REGION Network 1: Клапан регулирующий - 1
   // Зона - 1
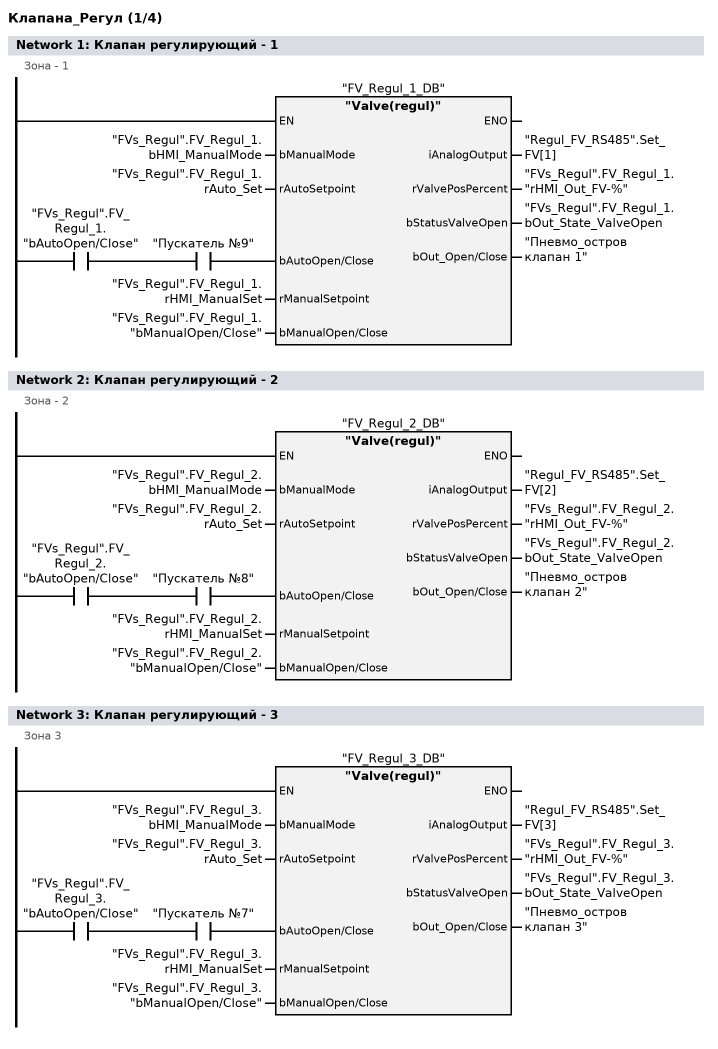
   RUNG wire#powerrail
      "FV_Regul_1_DB"("bAutoOpen/Close" := wire#w1, bManualMode := "FVs_Regul".FV_Regul_1.bHMI_ManualMode, rAutoSetpoint := "FVs_Regul".FV_Regul_1.rAuto_Set, rManualSetpoint := "FVs_Regul".FV_Regul_1.rHMI_ManualSet, "bManualOpen/Close" := "FVs_Regul".FV_Regul_1."bManualOpen/Close", iAnalogOutput => "Regul_FV_RS485".Set_FV[1], rValvePosPercent => "FVs_Regul".FV_Regul_1."rHMI_Out_FV-%", bStatusValveOpen => "FVs_Regul".FV_Regul_1.bOut_State_ValveOpen, "bOut_Open/Close" => "Пневмо_остров клапан 1")
   END_RUNG
   RUNG wire#powerrail
      Contact( "FVs_Regul".FV_Regul_1."bAutoOpen/Close" )
      Contact( "Пускатель №9" )
   END_RUNG wire#w1
   // the same network as SCL:
   "FV_Regul_1_DB"(bManualMode := "FVs_Regul".FV_Regul_1.bHMI_ManualMode,   // "Valve(regul)"
                   rAutoSetpoint := "FVs_Regul".FV_Regul_1.rAuto_Set,
                   "bAutoOpen/Close" := "FVs_Regul".FV_Regul_1."bAutoOpen/Close" AND "Пускатель №9",
                   rManualSetpoint := "FVs_Regul".FV_Regul_1.rHMI_ManualSet,
                   "bManualOpen/Close" := "FVs_Regul".FV_Regul_1."bManualOpen/Close",
                   iAnalogOutput => "Regul_FV_RS485".Set_FV[1],
                   rValvePosPercent => "FVs_Regul".FV_Regul_1."rHMI_Out_FV-%",
                   bStatusValveOpen => "FVs_Regul".FV_Regul_1.bOut_State_ValveOpen,
                   "bOut_Open/Close" => "Пневмо_остров клапан 1");
END_REGION

REGION Network 2: Клапан регулирующий - 2
   // Зона - 2
   RUNG wire#powerrail
      "FV_Regul_2_DB"("bAutoOpen/Close" := wire#w1, bManualMode := "FVs_Regul".FV_Regul_2.bHMI_ManualMode, rAutoSetpoint := "FVs_Regul".FV_Regul_2.rAuto_Set, rManualSetpoint := "FVs_Regul".FV_Regul_2.rHMI_ManualSet, "bManualOpen/Close" := "FVs_Regul".FV_Regul_2."bManualOpen/Close", iAnalogOutput => "Regul_FV_RS485".Set_FV[2], rValvePosPercent => "FVs_Regul".FV_Regul_2."rHMI_Out_FV-%", bStatusValveOpen => "FVs_Regul".FV_Regul_2.bOut_State_ValveOpen, "bOut_Open/Close" => "Пневмо_остров клапан 2")
   END_RUNG
   RUNG wire#powerrail
      Contact( "FVs_Regul".FV_Regul_2."bAutoOpen/Close" )
      Contact( "Пускатель №8" )
   END_RUNG wire#w1
   // the same network as SCL:
   "FV_Regul_2_DB"(bManualMode := "FVs_Regul".FV_Regul_2.bHMI_ManualMode,   // "Valve(regul)"
                   rAutoSetpoint := "FVs_Regul".FV_Regul_2.rAuto_Set,
                   "bAutoOpen/Close" := "FVs_Regul".FV_Regul_2."bAutoOpen/Close" AND "Пускатель №8",
                   rManualSetpoint := "FVs_Regul".FV_Regul_2.rHMI_ManualSet,
                   "bManualOpen/Close" := "FVs_Regul".FV_Regul_2."bManualOpen/Close",
                   iAnalogOutput => "Regul_FV_RS485".Set_FV[2],
                   rValvePosPercent => "FVs_Regul".FV_Regul_2."rHMI_Out_FV-%",
                   bStatusValveOpen => "FVs_Regul".FV_Regul_2.bOut_State_ValveOpen,
                   "bOut_Open/Close" => "Пневмо_остров клапан 2");
END_REGION

REGION Network 3: Клапан регулирующий - 3
   // Зона 3
   RUNG wire#powerrail
      "FV_Regul_3_DB"("bAutoOpen/Close" := wire#w1, bManualMode := "FVs_Regul".FV_Regul_3.bHMI_ManualMode, rAutoSetpoint := "FVs_Regul".FV_Regul_3.rAuto_Set, rManualSetpoint := "FVs_Regul".FV_Regul_3.rHMI_ManualSet, "bManualOpen/Close" := "FVs_Regul".FV_Regul_3."bManualOpen/Close", iAnalogOutput => "Regul_FV_RS485".Set_FV[3], rValvePosPercent => "FVs_Regul".FV_Regul_3."rHMI_Out_FV-%", bStatusValveOpen => "FVs_Regul".FV_Regul_3.bOut_State_ValveOpen, "bOut_Open/Close" => "Пневмо_остров клапан 3")
   END_RUNG
   RUNG wire#powerrail
      Contact( "FVs_Regul".FV_Regul_3."bAutoOpen/Close" )
      Contact( "Пускатель №7" )
   END_RUNG wire#w1
   // the same network as SCL:
   "FV_Regul_3_DB"(bManualMode := "FVs_Regul".FV_Regul_3.bHMI_ManualMode,   // "Valve(regul)"
                   rAutoSetpoint := "FVs_Regul".FV_Regul_3.rAuto_Set,
                   "bAutoOpen/Close" := "FVs_Regul".FV_Regul_3."bAutoOpen/Close" AND "Пускатель №7",
                   rManualSetpoint := "FVs_Regul".FV_Regul_3.rHMI_ManualSet,
                   "bManualOpen/Close" := "FVs_Regul".FV_Regul_3."bManualOpen/Close",
                   iAnalogOutput => "Regul_FV_RS485".Set_FV[3],
                   rValvePosPercent => "FVs_Regul".FV_Regul_3."rHMI_Out_FV-%",
                   bStatusValveOpen => "FVs_Regul".FV_Regul_3.bOut_State_ValveOpen,
                   "bOut_Open/Close" => "Пневмо_остров клапан 3");
END_REGION

REGION Network 4: Клапан регулирующий - 4
   // Зона 4
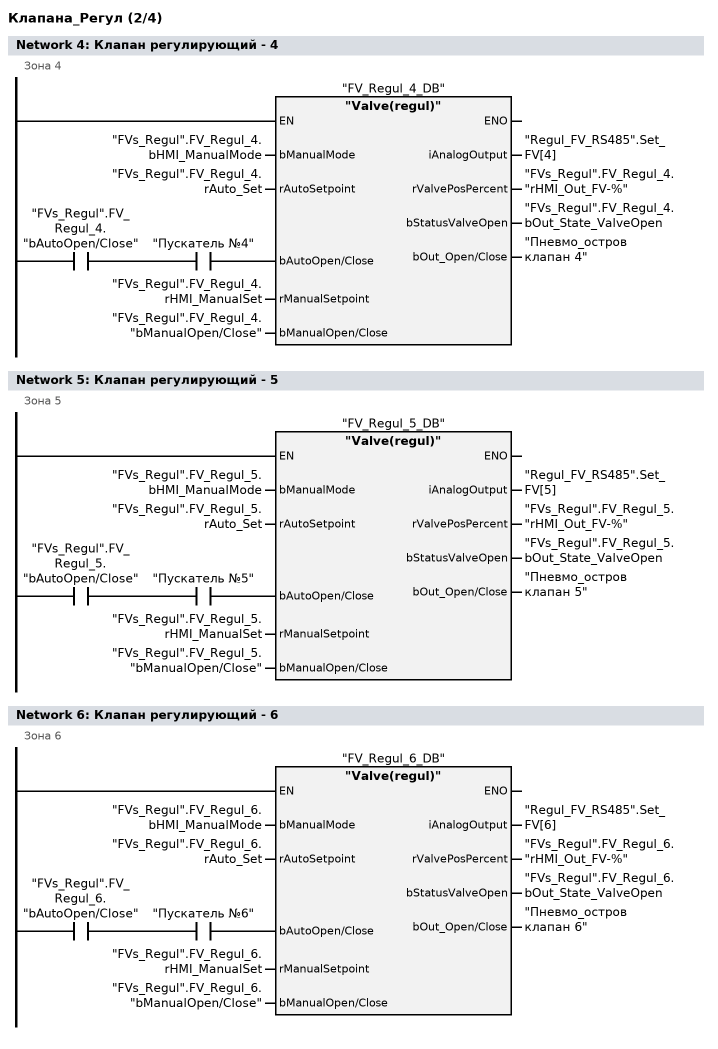
   RUNG wire#powerrail
      "FV_Regul_4_DB"("bAutoOpen/Close" := wire#w1, bManualMode := "FVs_Regul".FV_Regul_4.bHMI_ManualMode, rAutoSetpoint := "FVs_Regul".FV_Regul_4.rAuto_Set, rManualSetpoint := "FVs_Regul".FV_Regul_4.rHMI_ManualSet, "bManualOpen/Close" := "FVs_Regul".FV_Regul_4."bManualOpen/Close", iAnalogOutput => "Regul_FV_RS485".Set_FV[4], rValvePosPercent => "FVs_Regul".FV_Regul_4."rHMI_Out_FV-%", bStatusValveOpen => "FVs_Regul".FV_Regul_4.bOut_State_ValveOpen, "bOut_Open/Close" => "Пневмо_остров клапан 4")
   END_RUNG
   RUNG wire#powerrail
      Contact( "FVs_Regul".FV_Regul_4."bAutoOpen/Close" )
      Contact( "Пускатель №4" )
   END_RUNG wire#w1
   // the same network as SCL:
   "FV_Regul_4_DB"(bManualMode := "FVs_Regul".FV_Regul_4.bHMI_ManualMode,   // "Valve(regul)"
                   rAutoSetpoint := "FVs_Regul".FV_Regul_4.rAuto_Set,
                   "bAutoOpen/Close" := "FVs_Regul".FV_Regul_4."bAutoOpen/Close" AND "Пускатель №4",
                   rManualSetpoint := "FVs_Regul".FV_Regul_4.rHMI_ManualSet,
                   "bManualOpen/Close" := "FVs_Regul".FV_Regul_4."bManualOpen/Close",
                   iAnalogOutput => "Regul_FV_RS485".Set_FV[4],
                   rValvePosPercent => "FVs_Regul".FV_Regul_4."rHMI_Out_FV-%",
                   bStatusValveOpen => "FVs_Regul".FV_Regul_4.bOut_State_ValveOpen,
                   "bOut_Open/Close" => "Пневмо_остров клапан 4");
END_REGION

REGION Network 5: Клапан регулирующий - 5
   // Зона 5
   RUNG wire#powerrail
      "FV_Regul_5_DB"("bAutoOpen/Close" := wire#w1, bManualMode := "FVs_Regul".FV_Regul_5.bHMI_ManualMode, rAutoSetpoint := "FVs_Regul".FV_Regul_5.rAuto_Set, rManualSetpoint := "FVs_Regul".FV_Regul_5.rHMI_ManualSet, "bManualOpen/Close" := "FVs_Regul".FV_Regul_5."bManualOpen/Close", iAnalogOutput => "Regul_FV_RS485".Set_FV[5], rValvePosPercent => "FVs_Regul".FV_Regul_5."rHMI_Out_FV-%", bStatusValveOpen => "FVs_Regul".FV_Regul_5.bOut_State_ValveOpen, "bOut_Open/Close" => "Пневмо_остров клапан 5")
   END_RUNG
   RUNG wire#powerrail
      Contact( "FVs_Regul".FV_Regul_5."bAutoOpen/Close" )
      Contact( "Пускатель №5" )
   END_RUNG wire#w1
   // the same network as SCL:
   "FV_Regul_5_DB"(bManualMode := "FVs_Regul".FV_Regul_5.bHMI_ManualMode,   // "Valve(regul)"
                   rAutoSetpoint := "FVs_Regul".FV_Regul_5.rAuto_Set,
                   "bAutoOpen/Close" := "FVs_Regul".FV_Regul_5."bAutoOpen/Close" AND "Пускатель №5",
                   rManualSetpoint := "FVs_Regul".FV_Regul_5.rHMI_ManualSet,
                   "bManualOpen/Close" := "FVs_Regul".FV_Regul_5."bManualOpen/Close",
                   iAnalogOutput => "Regul_FV_RS485".Set_FV[5],
                   rValvePosPercent => "FVs_Regul".FV_Regul_5."rHMI_Out_FV-%",
                   bStatusValveOpen => "FVs_Regul".FV_Regul_5.bOut_State_ValveOpen,
                   "bOut_Open/Close" => "Пневмо_остров клапан 5");
END_REGION

REGION Network 6: Клапан регулирующий - 6
   // Зона 6
   RUNG wire#powerrail
      "FV_Regul_6_DB"("bAutoOpen/Close" := wire#w1, bManualMode := "FVs_Regul".FV_Regul_6.bHMI_ManualMode, rAutoSetpoint := "FVs_Regul".FV_Regul_6.rAuto_Set, rManualSetpoint := "FVs_Regul".FV_Regul_6.rHMI_ManualSet, "bManualOpen/Close" := "FVs_Regul".FV_Regul_6."bManualOpen/Close", iAnalogOutput => "Regul_FV_RS485".Set_FV[6], rValvePosPercent => "FVs_Regul".FV_Regul_6."rHMI_Out_FV-%", bStatusValveOpen => "FVs_Regul".FV_Regul_6.bOut_State_ValveOpen, "bOut_Open/Close" => "Пневмо_остров клапан 6")
   END_RUNG
   RUNG wire#powerrail
      Contact( "FVs_Regul".FV_Regul_6."bAutoOpen/Close" )
      Contact( "Пускатель №6" )
   END_RUNG wire#w1
   // the same network as SCL:
   "FV_Regul_6_DB"(bManualMode := "FVs_Regul".FV_Regul_6.bHMI_ManualMode,   // "Valve(regul)"
                   rAutoSetpoint := "FVs_Regul".FV_Regul_6.rAuto_Set,
                   "bAutoOpen/Close" := "FVs_Regul".FV_Regul_6."bAutoOpen/Close" AND "Пускатель №6",
                   rManualSetpoint := "FVs_Regul".FV_Regul_6.rHMI_ManualSet,
                   "bManualOpen/Close" := "FVs_Regul".FV_Regul_6."bManualOpen/Close",
                   iAnalogOutput => "Regul_FV_RS485".Set_FV[6],
                   rValvePosPercent => "FVs_Regul".FV_Regul_6."rHMI_Out_FV-%",
                   bStatusValveOpen => "FVs_Regul".FV_Regul_6.bOut_State_ValveOpen,
                   "bOut_Open/Close" => "Пневмо_остров клапан 6");
END_REGION

REGION Network 7: Клапан регулирующий - 7(Холод)
   // Зона 10 - Холод
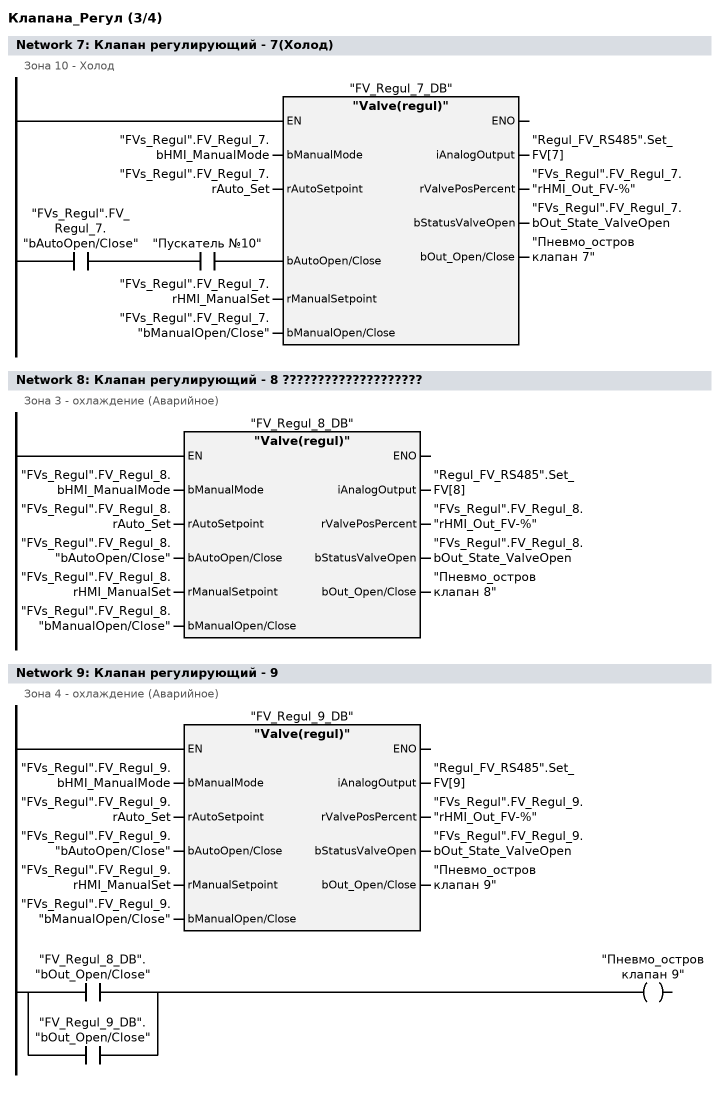
   RUNG wire#powerrail
      "FV_Regul_7_DB"("bAutoOpen/Close" := wire#w1, bManualMode := "FVs_Regul".FV_Regul_7.bHMI_ManualMode, rAutoSetpoint := "FVs_Regul".FV_Regul_7.rAuto_Set, rManualSetpoint := "FVs_Regul".FV_Regul_7.rHMI_ManualSet, "bManualOpen/Close" := "FVs_Regul".FV_Regul_7."bManualOpen/Close", iAnalogOutput => "Regul_FV_RS485".Set_FV[7], rValvePosPercent => "FVs_Regul".FV_Regul_7."rHMI_Out_FV-%", bStatusValveOpen => "FVs_Regul".FV_Regul_7.bOut_State_ValveOpen, "bOut_Open/Close" => "Пневмо_остров клапан 7")
   END_RUNG
   RUNG wire#powerrail
      Contact( "FVs_Regul".FV_Regul_7."bAutoOpen/Close" )
      Contact( "Пускатель №10" )
   END_RUNG wire#w1
   // the same network as SCL:
   "FV_Regul_7_DB"(bManualMode := "FVs_Regul".FV_Regul_7.bHMI_ManualMode,   // "Valve(regul)"
                   rAutoSetpoint := "FVs_Regul".FV_Regul_7.rAuto_Set,
                   "bAutoOpen/Close" := "FVs_Regul".FV_Regul_7."bAutoOpen/Close" AND "Пускатель №10",
                   rManualSetpoint := "FVs_Regul".FV_Regul_7.rHMI_ManualSet,
                   "bManualOpen/Close" := "FVs_Regul".FV_Regul_7."bManualOpen/Close",
                   iAnalogOutput => "Regul_FV_RS485".Set_FV[7],
                   rValvePosPercent => "FVs_Regul".FV_Regul_7."rHMI_Out_FV-%",
                   bStatusValveOpen => "FVs_Regul".FV_Regul_7.bOut_State_ValveOpen,
                   "bOut_Open/Close" => "Пневмо_остров клапан 7");
END_REGION

REGION Network 8: Клапан регулирующий - 8 ????????????????????
   // Зона 3 - охлаждение (Аварийное)
   RUNG wire#powerrail
      "FV_Regul_8_DB"(bManualMode := "FVs_Regul".FV_Regul_8.bHMI_ManualMode, rAutoSetpoint := "FVs_Regul".FV_Regul_8.rAuto_Set, "bAutoOpen/Close" := "FVs_Regul".FV_Regul_8."bAutoOpen/Close", rManualSetpoint := "FVs_Regul".FV_Regul_8.rHMI_ManualSet, "bManualOpen/Close" := "FVs_Regul".FV_Regul_8."bManualOpen/Close", iAnalogOutput => "Regul_FV_RS485".Set_FV[8], rValvePosPercent => "FVs_Regul".FV_Regul_8."rHMI_Out_FV-%", bStatusValveOpen => "FVs_Regul".FV_Regul_8.bOut_State_ValveOpen, "bOut_Open/Close" => "Пневмо_остров клапан 8")
   END_RUNG
   // the same network as SCL:
   "FV_Regul_8_DB"(bManualMode := "FVs_Regul".FV_Regul_8.bHMI_ManualMode,   // "Valve(regul)"
                   rAutoSetpoint := "FVs_Regul".FV_Regul_8.rAuto_Set,
                   "bAutoOpen/Close" := "FVs_Regul".FV_Regul_8."bAutoOpen/Close",
                   rManualSetpoint := "FVs_Regul".FV_Regul_8.rHMI_ManualSet,
                   "bManualOpen/Close" := "FVs_Regul".FV_Regul_8."bManualOpen/Close",
                   iAnalogOutput => "Regul_FV_RS485".Set_FV[8],
                   rValvePosPercent => "FVs_Regul".FV_Regul_8."rHMI_Out_FV-%",
                   bStatusValveOpen => "FVs_Regul".FV_Regul_8.bOut_State_ValveOpen,
                   "bOut_Open/Close" => "Пневмо_остров клапан 8");
END_REGION

REGION Network 9: Клапан регулирующий - 9
   // Зона 4 - охлаждение (Аварийное)
   RUNG wire#powerrail
      "FV_Regul_9_DB"(bManualMode := "FVs_Regul".FV_Regul_9.bHMI_ManualMode, rAutoSetpoint := "FVs_Regul".FV_Regul_9.rAuto_Set, "bAutoOpen/Close" := "FVs_Regul".FV_Regul_9."bAutoOpen/Close", rManualSetpoint := "FVs_Regul".FV_Regul_9.rHMI_ManualSet, "bManualOpen/Close" := "FVs_Regul".FV_Regul_9."bManualOpen/Close", iAnalogOutput => "Regul_FV_RS485".Set_FV[9], rValvePosPercent => "FVs_Regul".FV_Regul_9."rHMI_Out_FV-%", bStatusValveOpen => "FVs_Regul".FV_Regul_9.bOut_State_ValveOpen, "bOut_Open/Close" => "Пневмо_остров клапан 9")
   END_RUNG
   RUNG wire#powerrail
      Contact( "FV_Regul_8_DB"."bOut_Open/Close" )
      wire#w1
      Coil( "Пневмо_остров клапан 9" )
   END_RUNG
   RUNG wire#powerrail
      Contact( "FV_Regul_9_DB"."bOut_Open/Close" )
   END_RUNG wire#w1
   // the same network as SCL:
   "FV_Regul_9_DB"(bManualMode := "FVs_Regul".FV_Regul_9.bHMI_ManualMode,   // "Valve(regul)"
                   rAutoSetpoint := "FVs_Regul".FV_Regul_9.rAuto_Set,
                   "bAutoOpen/Close" := "FVs_Regul".FV_Regul_9."bAutoOpen/Close",
                   rManualSetpoint := "FVs_Regul".FV_Regul_9.rHMI_ManualSet,
                   "bManualOpen/Close" := "FVs_Regul".FV_Regul_9."bManualOpen/Close",
                   iAnalogOutput => "Regul_FV_RS485".Set_FV[9],
                   rValvePosPercent => "FVs_Regul".FV_Regul_9."rHMI_Out_FV-%",
                   bStatusValveOpen => "FVs_Regul".FV_Regul_9.bOut_State_ValveOpen,
                   "bOut_Open/Close" => "Пневмо_остров клапан 9");
   "Пневмо_остров клапан 9" := "FV_Regul_8_DB"."bOut_Open/Close" OR "FV_Regul_9_DB"."bOut_Open/Close";
END_REGION

REGION Network 10: Клапан регулирующий - 10
   // Зона 5 - охлаждение (аварийное)
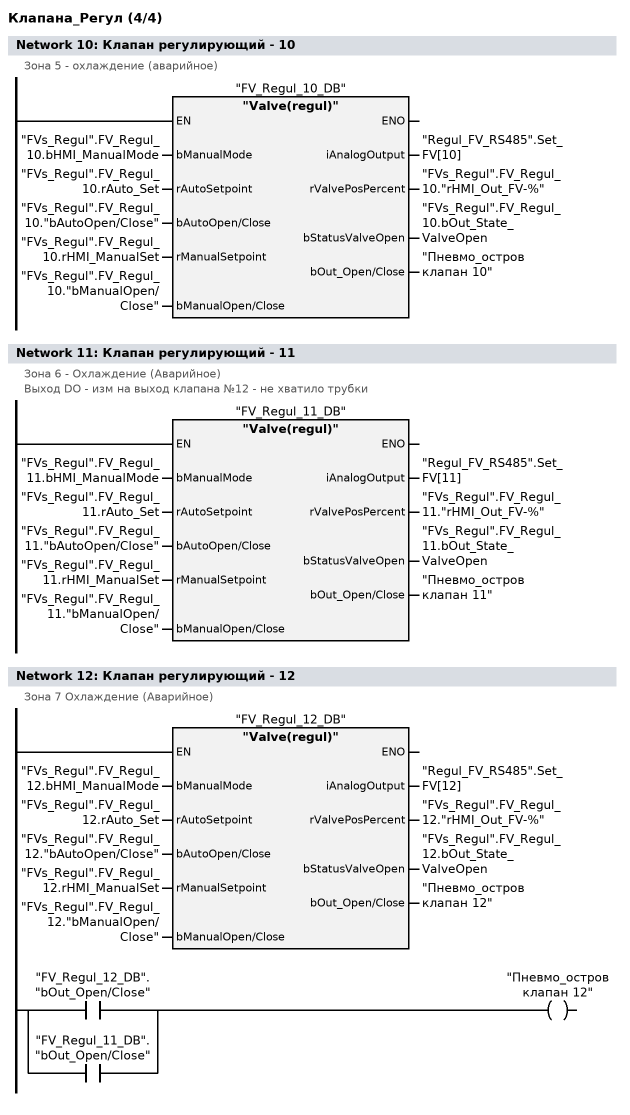
   RUNG wire#powerrail
      "FV_Regul_10_DB"(bManualMode := "FVs_Regul".FV_Regul_10.bHMI_ManualMode, rAutoSetpoint := "FVs_Regul".FV_Regul_10.rAuto_Set, "bAutoOpen/Close" := "FVs_Regul".FV_Regul_10."bAutoOpen/Close", rManualSetpoint := "FVs_Regul".FV_Regul_10.rHMI_ManualSet, "bManualOpen/Close" := "FVs_Regul".FV_Regul_10."bManualOpen/Close", iAnalogOutput => "Regul_FV_RS485".Set_FV[10], rValvePosPercent => "FVs_Regul".FV_Regul_10."rHMI_Out_FV-%", bStatusValveOpen => "FVs_Regul".FV_Regul_10.bOut_State_ValveOpen, "bOut_Open/Close" => "Пневмо_остров клапан 10")
   END_RUNG
   // the same network as SCL:
   "FV_Regul_10_DB"(bManualMode := "FVs_Regul".FV_Regul_10.bHMI_ManualMode,   // "Valve(regul)"
                    rAutoSetpoint := "FVs_Regul".FV_Regul_10.rAuto_Set,
                    "bAutoOpen/Close" := "FVs_Regul".FV_Regul_10."bAutoOpen/Close",
                    rManualSetpoint := "FVs_Regul".FV_Regul_10.rHMI_ManualSet,
                    "bManualOpen/Close" := "FVs_Regul".FV_Regul_10."bManualOpen/Close",
                    iAnalogOutput => "Regul_FV_RS485".Set_FV[10],
                    rValvePosPercent => "FVs_Regul".FV_Regul_10."rHMI_Out_FV-%",
                    bStatusValveOpen => "FVs_Regul".FV_Regul_10.bOut_State_ValveOpen,
                    "bOut_Open/Close" => "Пневмо_остров клапан 10");
END_REGION

REGION Network 11: Клапан регулирующий - 11
   // Зона 6 - Охлаждение (Аварийное)
   // Выход DO - изм на выход клапана №12 - не хватило трубки
   RUNG wire#powerrail
      "FV_Regul_11_DB"(bManualMode := "FVs_Regul".FV_Regul_11.bHMI_ManualMode, rAutoSetpoint := "FVs_Regul".FV_Regul_11.rAuto_Set, "bAutoOpen/Close" := "FVs_Regul".FV_Regul_11."bAutoOpen/Close", rManualSetpoint := "FVs_Regul".FV_Regul_11.rHMI_ManualSet, "bManualOpen/Close" := "FVs_Regul".FV_Regul_11."bManualOpen/Close", iAnalogOutput => "Regul_FV_RS485".Set_FV[11], rValvePosPercent => "FVs_Regul".FV_Regul_11."rHMI_Out_FV-%", bStatusValveOpen => "FVs_Regul".FV_Regul_11.bOut_State_ValveOpen, "bOut_Open/Close" => "Пневмо_остров клапан 11")
   END_RUNG
   // the same network as SCL:
   "FV_Regul_11_DB"(bManualMode := "FVs_Regul".FV_Regul_11.bHMI_ManualMode,   // "Valve(regul)"
                    rAutoSetpoint := "FVs_Regul".FV_Regul_11.rAuto_Set,
                    "bAutoOpen/Close" := "FVs_Regul".FV_Regul_11."bAutoOpen/Close",
                    rManualSetpoint := "FVs_Regul".FV_Regul_11.rHMI_ManualSet,
                    "bManualOpen/Close" := "FVs_Regul".FV_Regul_11."bManualOpen/Close",
                    iAnalogOutput => "Regul_FV_RS485".Set_FV[11],
                    rValvePosPercent => "FVs_Regul".FV_Regul_11."rHMI_Out_FV-%",
                    bStatusValveOpen => "FVs_Regul".FV_Regul_11.bOut_State_ValveOpen,
                    "bOut_Open/Close" => "Пневмо_остров клапан 11");
END_REGION

REGION Network 12: Клапан регулирующий - 12
   // Зона 7 Охлаждение (Аварийное)
   RUNG wire#powerrail
      "FV_Regul_12_DB"(bManualMode := "FVs_Regul".FV_Regul_12.bHMI_ManualMode, rAutoSetpoint := "FVs_Regul".FV_Regul_12.rAuto_Set, "bAutoOpen/Close" := "FVs_Regul".FV_Regul_12."bAutoOpen/Close", rManualSetpoint := "FVs_Regul".FV_Regul_12.rHMI_ManualSet, "bManualOpen/Close" := "FVs_Regul".FV_Regul_12."bManualOpen/Close", iAnalogOutput => "Regul_FV_RS485".Set_FV[12], rValvePosPercent => "FVs_Regul".FV_Regul_12."rHMI_Out_FV-%", bStatusValveOpen => "FVs_Regul".FV_Regul_12.bOut_State_ValveOpen, "bOut_Open/Close" => "Пневмо_остров клапан 12")
   END_RUNG
   RUNG wire#powerrail
      Contact( "FV_Regul_12_DB"."bOut_Open/Close" )
      wire#w1
      Coil( "Пневмо_остров клапан 12" )
   END_RUNG
   RUNG wire#powerrail
      Contact( "FV_Regul_11_DB"."bOut_Open/Close" )
   END_RUNG wire#w1
   // the same network as SCL:
   "FV_Regul_12_DB"(bManualMode := "FVs_Regul".FV_Regul_12.bHMI_ManualMode,   // "Valve(regul)"
                    rAutoSetpoint := "FVs_Regul".FV_Regul_12.rAuto_Set,
                    "bAutoOpen/Close" := "FVs_Regul".FV_Regul_12."bAutoOpen/Close",
                    rManualSetpoint := "FVs_Regul".FV_Regul_12.rHMI_ManualSet,
                    "bManualOpen/Close" := "FVs_Regul".FV_Regul_12."bManualOpen/Close",
                    iAnalogOutput => "Regul_FV_RS485".Set_FV[12],
                    rValvePosPercent => "FVs_Regul".FV_Regul_12."rHMI_Out_FV-%",
                    bStatusValveOpen => "FVs_Regul".FV_Regul_12.bOut_State_ValveOpen,
                    "bOut_Open/Close" => "Пневмо_остров клапан 12");
   "Пневмо_остров клапан 12" := "FV_Regul_12_DB"."bOut_Open/Close" OR "FV_Regul_11_DB"."bOut_Open/Close";
END_REGION

REGION Network 13 (SCL): Клапана регулирующие ручной режим с вфходом DO
   // Для перевода клапана регулирующего в ручной режим должен перейти по сигналу от ручного режим с клапана DO, т.е. для работы клапана регулирующего необходим сигнал DO
   (*"FVs_o/p".FV_1.bManualMode := "FVs_Regul".FV_Regul_1.bHMI_ManualMode;
   "FVs_o/p".FV_2.bManualMode := "FVs_Regul".FV_Regul_2.bHMI_ManualMode;
   "FVs_o/p".FV_3.bManualMode := "FVs_Regul".FV_Regul_3.bHMI_ManualMode;
   "FVs_o/p".FV_4.bManualMode := "FVs_Regul".FV_Regul_5.bHMI_ManualMode;
   *)
END_REGION
END_FUNCTION

FUNCTION "Зоны Пастеризации_Контроль" : Void   // FC3, LAD
{ S7_Optimized_Access := 'TRUE' }
VERSION : 0.1
BEGIN

REGION Network 1: Зона 1(Нагрев)
   // Зона 1
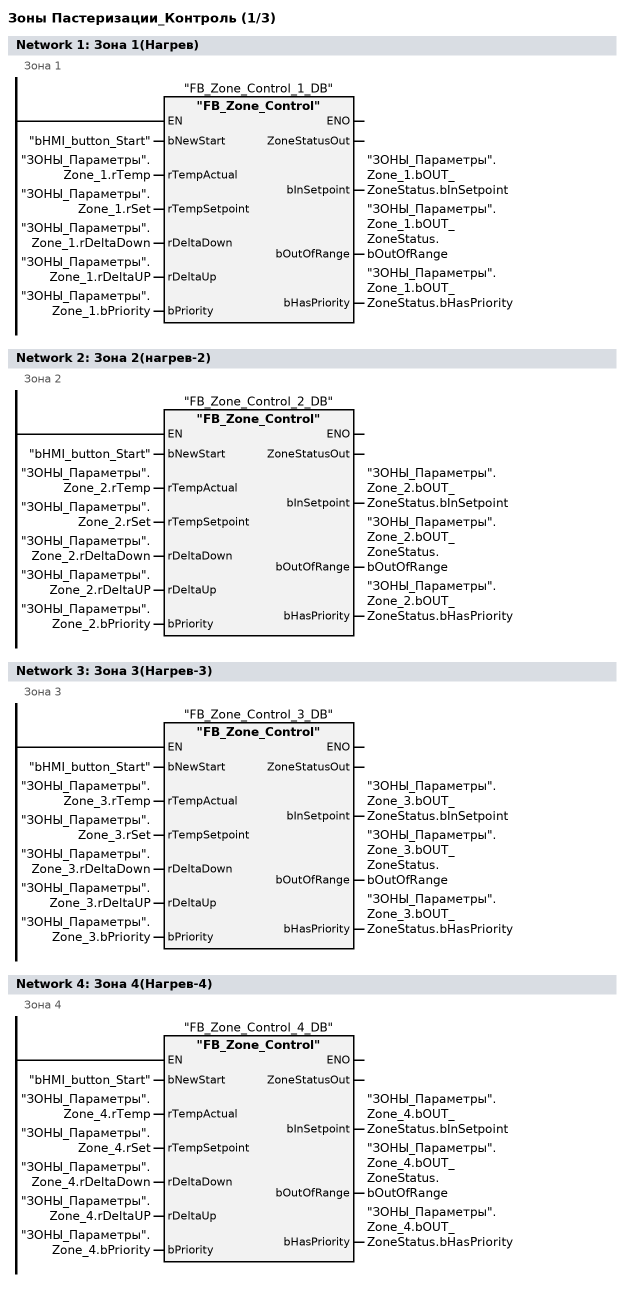
   RUNG wire#powerrail
      "FB_Zone_Control_1_DB"(bNewStart := "bHMI_button_Start", rTempActual := "ЗОНЫ_Параметры".Zone_1.rTemp, rTempSetpoint := "ЗОНЫ_Параметры".Zone_1.rSet, rDeltaDown := "ЗОНЫ_Параметры".Zone_1.rDeltaDown, rDeltaUp := "ЗОНЫ_Параметры".Zone_1.rDeltaUP, bPriority := "ЗОНЫ_Параметры".Zone_1.bPriority, ZoneStatusOut =>, bInSetpoint => "ЗОНЫ_Параметры".Zone_1.bOUT_ZoneStatus.bInSetpoint, bOutOfRange => "ЗОНЫ_Параметры".Zone_1.bOUT_ZoneStatus.bOutOfRange, bHasPriority => "ЗОНЫ_Параметры".Zone_1.bOUT_ZoneStatus.bHasPriority)
   END_RUNG
   // the same network as SCL:
   "FB_Zone_Control_1_DB"(bNewStart := "bHMI_button_Start",   // "FB_Zone_Control"
                          rTempActual := "ЗОНЫ_Параметры".Zone_1.rTemp,
                          rTempSetpoint := "ЗОНЫ_Параметры".Zone_1.rSet,
                          rDeltaDown := "ЗОНЫ_Параметры".Zone_1.rDeltaDown,
                          rDeltaUp := "ЗОНЫ_Параметры".Zone_1.rDeltaUP,
                          bPriority := "ЗОНЫ_Параметры".Zone_1.bPriority,
                          bInSetpoint => "ЗОНЫ_Параметры".Zone_1.bOUT_ZoneStatus.bInSetpoint,
                          bOutOfRange => "ЗОНЫ_Параметры".Zone_1.bOUT_ZoneStatus.bOutOfRange,
                          bHasPriority => "ЗОНЫ_Параметры".Zone_1.bOUT_ZoneStatus.bHasPriority);
END_REGION

REGION Network 2: Зона 2(нагрев-2)
   // Зона 2
   RUNG wire#powerrail
      "FB_Zone_Control_2_DB"(bNewStart := "bHMI_button_Start", rTempActual := "ЗОНЫ_Параметры".Zone_2.rTemp, rTempSetpoint := "ЗОНЫ_Параметры".Zone_2.rSet, rDeltaDown := "ЗОНЫ_Параметры".Zone_2.rDeltaDown, rDeltaUp := "ЗОНЫ_Параметры".Zone_2.rDeltaUP, bPriority := "ЗОНЫ_Параметры".Zone_2.bPriority, ZoneStatusOut =>, bInSetpoint => "ЗОНЫ_Параметры".Zone_2.bOUT_ZoneStatus.bInSetpoint, bOutOfRange => "ЗОНЫ_Параметры".Zone_2.bOUT_ZoneStatus.bOutOfRange, bHasPriority => "ЗОНЫ_Параметры".Zone_2.bOUT_ZoneStatus.bHasPriority)
   END_RUNG
   // the same network as SCL:
   "FB_Zone_Control_2_DB"(bNewStart := "bHMI_button_Start",   // "FB_Zone_Control"
                          rTempActual := "ЗОНЫ_Параметры".Zone_2.rTemp,
                          rTempSetpoint := "ЗОНЫ_Параметры".Zone_2.rSet,
                          rDeltaDown := "ЗОНЫ_Параметры".Zone_2.rDeltaDown,
                          rDeltaUp := "ЗОНЫ_Параметры".Zone_2.rDeltaUP,
                          bPriority := "ЗОНЫ_Параметры".Zone_2.bPriority,
                          bInSetpoint => "ЗОНЫ_Параметры".Zone_2.bOUT_ZoneStatus.bInSetpoint,
                          bOutOfRange => "ЗОНЫ_Параметры".Zone_2.bOUT_ZoneStatus.bOutOfRange,
                          bHasPriority => "ЗОНЫ_Параметры".Zone_2.bOUT_ZoneStatus.bHasPriority);
END_REGION

REGION Network 3: Зона 3(Нагрев-3)
   // Зона 3
   RUNG wire#powerrail
      "FB_Zone_Control_3_DB"(bNewStart := "bHMI_button_Start", rTempActual := "ЗОНЫ_Параметры".Zone_3.rTemp, rTempSetpoint := "ЗОНЫ_Параметры".Zone_3.rSet, rDeltaDown := "ЗОНЫ_Параметры".Zone_3.rDeltaDown, rDeltaUp := "ЗОНЫ_Параметры".Zone_3.rDeltaUP, bPriority := "ЗОНЫ_Параметры".Zone_3.bPriority, ZoneStatusOut =>, bInSetpoint => "ЗОНЫ_Параметры".Zone_3.bOUT_ZoneStatus.bInSetpoint, bOutOfRange => "ЗОНЫ_Параметры".Zone_3.bOUT_ZoneStatus.bOutOfRange, bHasPriority => "ЗОНЫ_Параметры".Zone_3.bOUT_ZoneStatus.bHasPriority)
   END_RUNG
   // the same network as SCL:
   "FB_Zone_Control_3_DB"(bNewStart := "bHMI_button_Start",   // "FB_Zone_Control"
                          rTempActual := "ЗОНЫ_Параметры".Zone_3.rTemp,
                          rTempSetpoint := "ЗОНЫ_Параметры".Zone_3.rSet,
                          rDeltaDown := "ЗОНЫ_Параметры".Zone_3.rDeltaDown,
                          rDeltaUp := "ЗОНЫ_Параметры".Zone_3.rDeltaUP,
                          bPriority := "ЗОНЫ_Параметры".Zone_3.bPriority,
                          bInSetpoint => "ЗОНЫ_Параметры".Zone_3.bOUT_ZoneStatus.bInSetpoint,
                          bOutOfRange => "ЗОНЫ_Параметры".Zone_3.bOUT_ZoneStatus.bOutOfRange,
                          bHasPriority => "ЗОНЫ_Параметры".Zone_3.bOUT_ZoneStatus.bHasPriority);
END_REGION

REGION Network 4: Зона 4(Нагрев-4)
   // Зона 4
   RUNG wire#powerrail
      "FB_Zone_Control_4_DB"(bNewStart := "bHMI_button_Start", rTempActual := "ЗОНЫ_Параметры".Zone_4.rTemp, rTempSetpoint := "ЗОНЫ_Параметры".Zone_4.rSet, rDeltaDown := "ЗОНЫ_Параметры".Zone_4.rDeltaDown, rDeltaUp := "ЗОНЫ_Параметры".Zone_4.rDeltaUP, bPriority := "ЗОНЫ_Параметры".Zone_4.bPriority, ZoneStatusOut =>, bInSetpoint => "ЗОНЫ_Параметры".Zone_4.bOUT_ZoneStatus.bInSetpoint, bOutOfRange => "ЗОНЫ_Параметры".Zone_4.bOUT_ZoneStatus.bOutOfRange, bHasPriority => "ЗОНЫ_Параметры".Zone_4.bOUT_ZoneStatus.bHasPriority)
   END_RUNG
   // the same network as SCL:
   "FB_Zone_Control_4_DB"(bNewStart := "bHMI_button_Start",   // "FB_Zone_Control"
                          rTempActual := "ЗОНЫ_Параметры".Zone_4.rTemp,
                          rTempSetpoint := "ЗОНЫ_Параметры".Zone_4.rSet,
                          rDeltaDown := "ЗОНЫ_Параметры".Zone_4.rDeltaDown,
                          rDeltaUp := "ЗОНЫ_Параметры".Zone_4.rDeltaUP,
                          bPriority := "ЗОНЫ_Параметры".Zone_4.bPriority,
                          bInSetpoint => "ЗОНЫ_Параметры".Zone_4.bOUT_ZoneStatus.bInSetpoint,
                          bOutOfRange => "ЗОНЫ_Параметры".Zone_4.bOUT_ZoneStatus.bOutOfRange,
                          bHasPriority => "ЗОНЫ_Параметры".Zone_4.bOUT_ZoneStatus.bHasPriority);
END_REGION

REGION Network 5: Зона 5(Выдержка-1)
   // Зона 5
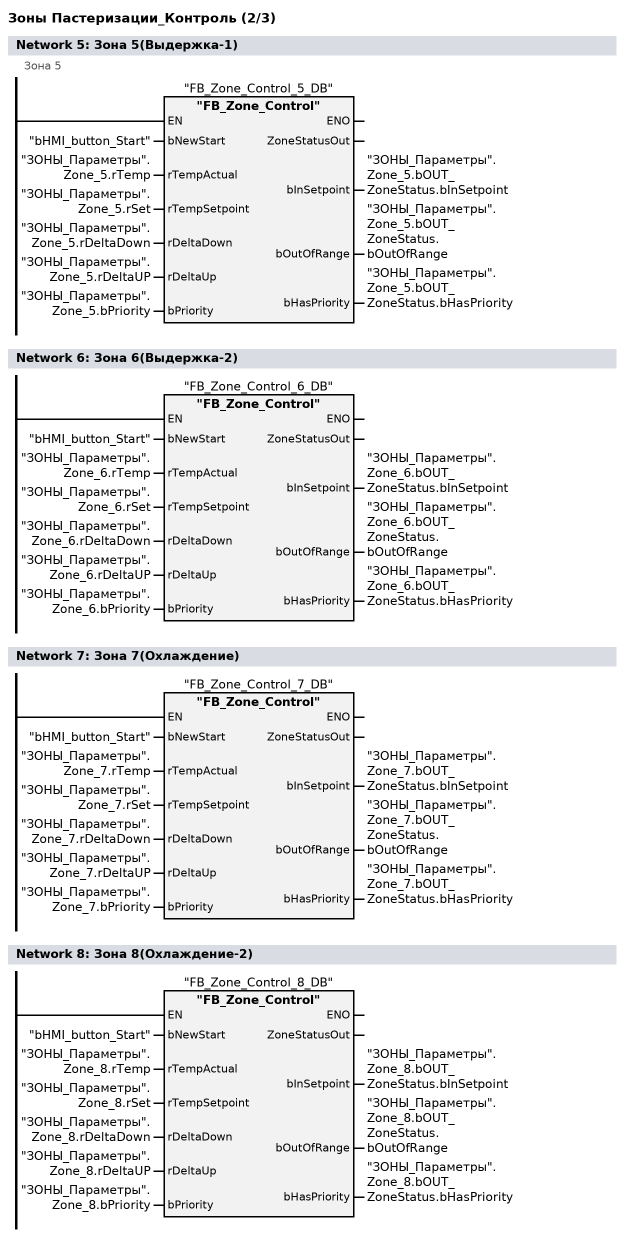
   RUNG wire#powerrail
      "FB_Zone_Control_5_DB"(bNewStart := "bHMI_button_Start", rTempActual := "ЗОНЫ_Параметры".Zone_5.rTemp, rTempSetpoint := "ЗОНЫ_Параметры".Zone_5.rSet, rDeltaDown := "ЗОНЫ_Параметры".Zone_5.rDeltaDown, rDeltaUp := "ЗОНЫ_Параметры".Zone_5.rDeltaUP, bPriority := "ЗОНЫ_Параметры".Zone_5.bPriority, ZoneStatusOut =>, bInSetpoint => "ЗОНЫ_Параметры".Zone_5.bOUT_ZoneStatus.bInSetpoint, bOutOfRange => "ЗОНЫ_Параметры".Zone_5.bOUT_ZoneStatus.bOutOfRange, bHasPriority => "ЗОНЫ_Параметры".Zone_5.bOUT_ZoneStatus.bHasPriority)
   END_RUNG
   // the same network as SCL:
   "FB_Zone_Control_5_DB"(bNewStart := "bHMI_button_Start",   // "FB_Zone_Control"
                          rTempActual := "ЗОНЫ_Параметры".Zone_5.rTemp,
                          rTempSetpoint := "ЗОНЫ_Параметры".Zone_5.rSet,
                          rDeltaDown := "ЗОНЫ_Параметры".Zone_5.rDeltaDown,
                          rDeltaUp := "ЗОНЫ_Параметры".Zone_5.rDeltaUP,
                          bPriority := "ЗОНЫ_Параметры".Zone_5.bPriority,
                          bInSetpoint => "ЗОНЫ_Параметры".Zone_5.bOUT_ZoneStatus.bInSetpoint,
                          bOutOfRange => "ЗОНЫ_Параметры".Zone_5.bOUT_ZoneStatus.bOutOfRange,
                          bHasPriority => "ЗОНЫ_Параметры".Zone_5.bOUT_ZoneStatus.bHasPriority);
END_REGION

REGION Network 6: Зона 6(Выдержка-2)
   RUNG wire#powerrail
      "FB_Zone_Control_6_DB"(bNewStart := "bHMI_button_Start", rTempActual := "ЗОНЫ_Параметры".Zone_6.rTemp, rTempSetpoint := "ЗОНЫ_Параметры".Zone_6.rSet, rDeltaDown := "ЗОНЫ_Параметры".Zone_6.rDeltaDown, rDeltaUp := "ЗОНЫ_Параметры".Zone_6.rDeltaUP, bPriority := "ЗОНЫ_Параметры".Zone_6.bPriority, ZoneStatusOut =>, bInSetpoint => "ЗОНЫ_Параметры".Zone_6.bOUT_ZoneStatus.bInSetpoint, bOutOfRange => "ЗОНЫ_Параметры".Zone_6.bOUT_ZoneStatus.bOutOfRange, bHasPriority => "ЗОНЫ_Параметры".Zone_6.bOUT_ZoneStatus.bHasPriority)
   END_RUNG
   // the same network as SCL:
   "FB_Zone_Control_6_DB"(bNewStart := "bHMI_button_Start",   // "FB_Zone_Control"
                          rTempActual := "ЗОНЫ_Параметры".Zone_6.rTemp,
                          rTempSetpoint := "ЗОНЫ_Параметры".Zone_6.rSet,
                          rDeltaDown := "ЗОНЫ_Параметры".Zone_6.rDeltaDown,
                          rDeltaUp := "ЗОНЫ_Параметры".Zone_6.rDeltaUP,
                          bPriority := "ЗОНЫ_Параметры".Zone_6.bPriority,
                          bInSetpoint => "ЗОНЫ_Параметры".Zone_6.bOUT_ZoneStatus.bInSetpoint,
                          bOutOfRange => "ЗОНЫ_Параметры".Zone_6.bOUT_ZoneStatus.bOutOfRange,
                          bHasPriority => "ЗОНЫ_Параметры".Zone_6.bOUT_ZoneStatus.bHasPriority);
END_REGION

REGION Network 7: Зона 7(Охлаждение)
   RUNG wire#powerrail
      "FB_Zone_Control_7_DB"(bNewStart := "bHMI_button_Start", rTempActual := "ЗОНЫ_Параметры".Zone_7.rTemp, rTempSetpoint := "ЗОНЫ_Параметры".Zone_7.rSet, rDeltaDown := "ЗОНЫ_Параметры".Zone_7.rDeltaDown, rDeltaUp := "ЗОНЫ_Параметры".Zone_7.rDeltaUP, bPriority := "ЗОНЫ_Параметры".Zone_7.bPriority, ZoneStatusOut =>, bInSetpoint => "ЗОНЫ_Параметры".Zone_7.bOUT_ZoneStatus.bInSetpoint, bOutOfRange => "ЗОНЫ_Параметры".Zone_7.bOUT_ZoneStatus.bOutOfRange, bHasPriority => "ЗОНЫ_Параметры".Zone_7.bOUT_ZoneStatus.bHasPriority)
   END_RUNG
   // the same network as SCL:
   "FB_Zone_Control_7_DB"(bNewStart := "bHMI_button_Start",   // "FB_Zone_Control"
                          rTempActual := "ЗОНЫ_Параметры".Zone_7.rTemp,
                          rTempSetpoint := "ЗОНЫ_Параметры".Zone_7.rSet,
                          rDeltaDown := "ЗОНЫ_Параметры".Zone_7.rDeltaDown,
                          rDeltaUp := "ЗОНЫ_Параметры".Zone_7.rDeltaUP,
                          bPriority := "ЗОНЫ_Параметры".Zone_7.bPriority,
                          bInSetpoint => "ЗОНЫ_Параметры".Zone_7.bOUT_ZoneStatus.bInSetpoint,
                          bOutOfRange => "ЗОНЫ_Параметры".Zone_7.bOUT_ZoneStatus.bOutOfRange,
                          bHasPriority => "ЗОНЫ_Параметры".Zone_7.bOUT_ZoneStatus.bHasPriority);
END_REGION

REGION Network 8: Зона 8(Охлаждение-2)
   RUNG wire#powerrail
      "FB_Zone_Control_8_DB"(bNewStart := "bHMI_button_Start", rTempActual := "ЗОНЫ_Параметры".Zone_8.rTemp, rTempSetpoint := "ЗОНЫ_Параметры".Zone_8.rSet, rDeltaDown := "ЗОНЫ_Параметры".Zone_8.rDeltaDown, rDeltaUp := "ЗОНЫ_Параметры".Zone_8.rDeltaUP, bPriority := "ЗОНЫ_Параметры".Zone_8.bPriority, ZoneStatusOut =>, bInSetpoint => "ЗОНЫ_Параметры".Zone_8.bOUT_ZoneStatus.bInSetpoint, bOutOfRange => "ЗОНЫ_Параметры".Zone_8.bOUT_ZoneStatus.bOutOfRange, bHasPriority => "ЗОНЫ_Параметры".Zone_8.bOUT_ZoneStatus.bHasPriority)
   END_RUNG
   // the same network as SCL:
   "FB_Zone_Control_8_DB"(bNewStart := "bHMI_button_Start",   // "FB_Zone_Control"
                          rTempActual := "ЗОНЫ_Параметры".Zone_8.rTemp,
                          rTempSetpoint := "ЗОНЫ_Параметры".Zone_8.rSet,
                          rDeltaDown := "ЗОНЫ_Параметры".Zone_8.rDeltaDown,
                          rDeltaUp := "ЗОНЫ_Параметры".Zone_8.rDeltaUP,
                          bPriority := "ЗОНЫ_Параметры".Zone_8.bPriority,
                          bInSetpoint => "ЗОНЫ_Параметры".Zone_8.bOUT_ZoneStatus.bInSetpoint,
                          bOutOfRange => "ЗОНЫ_Параметры".Zone_8.bOUT_ZoneStatus.bOutOfRange,
                          bHasPriority => "ЗОНЫ_Параметры".Zone_8.bOUT_ZoneStatus.bHasPriority);
END_REGION

REGION Network 9: Зона 9(Охлаждение-3)
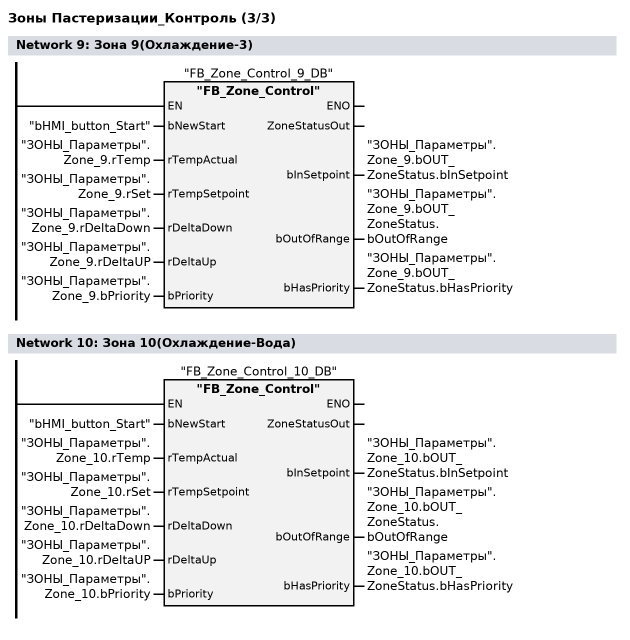
   RUNG wire#powerrail
      "FB_Zone_Control_9_DB"(bNewStart := "bHMI_button_Start", rTempActual := "ЗОНЫ_Параметры".Zone_9.rTemp, rTempSetpoint := "ЗОНЫ_Параметры".Zone_9.rSet, rDeltaDown := "ЗОНЫ_Параметры".Zone_9.rDeltaDown, rDeltaUp := "ЗОНЫ_Параметры".Zone_9.rDeltaUP, bPriority := "ЗОНЫ_Параметры".Zone_9.bPriority, ZoneStatusOut =>, bInSetpoint => "ЗОНЫ_Параметры".Zone_9.bOUT_ZoneStatus.bInSetpoint, bOutOfRange => "ЗОНЫ_Параметры".Zone_9.bOUT_ZoneStatus.bOutOfRange, bHasPriority => "ЗОНЫ_Параметры".Zone_9.bOUT_ZoneStatus.bHasPriority)
   END_RUNG
   // the same network as SCL:
   "FB_Zone_Control_9_DB"(bNewStart := "bHMI_button_Start",   // "FB_Zone_Control"
                          rTempActual := "ЗОНЫ_Параметры".Zone_9.rTemp,
                          rTempSetpoint := "ЗОНЫ_Параметры".Zone_9.rSet,
                          rDeltaDown := "ЗОНЫ_Параметры".Zone_9.rDeltaDown,
                          rDeltaUp := "ЗОНЫ_Параметры".Zone_9.rDeltaUP,
                          bPriority := "ЗОНЫ_Параметры".Zone_9.bPriority,
                          bInSetpoint => "ЗОНЫ_Параметры".Zone_9.bOUT_ZoneStatus.bInSetpoint,
                          bOutOfRange => "ЗОНЫ_Параметры".Zone_9.bOUT_ZoneStatus.bOutOfRange,
                          bHasPriority => "ЗОНЫ_Параметры".Zone_9.bOUT_ZoneStatus.bHasPriority);
END_REGION

REGION Network 10: Зона 10(Охлаждение-Вода)
   RUNG wire#powerrail
      "FB_Zone_Control_10_DB"(bNewStart := "bHMI_button_Start", rTempActual := "ЗОНЫ_Параметры".Zone_10.rTemp, rTempSetpoint := "ЗОНЫ_Параметры".Zone_10.rSet, rDeltaDown := "ЗОНЫ_Параметры".Zone_10.rDeltaDown, rDeltaUp := "ЗОНЫ_Параметры".Zone_10.rDeltaUP, bPriority := "ЗОНЫ_Параметры".Zone_10.bPriority, ZoneStatusOut =>, bInSetpoint => "ЗОНЫ_Параметры".Zone_10.bOUT_ZoneStatus.bInSetpoint, bOutOfRange => "ЗОНЫ_Параметры".Zone_10.bOUT_ZoneStatus.bOutOfRange, bHasPriority => "ЗОНЫ_Параметры".Zone_10.bOUT_ZoneStatus.bHasPriority)
   END_RUNG
   // the same network as SCL:
   "FB_Zone_Control_10_DB"(bNewStart := "bHMI_button_Start",   // "FB_Zone_Control"
                           rTempActual := "ЗОНЫ_Параметры".Zone_10.rTemp,
                           rTempSetpoint := "ЗОНЫ_Параметры".Zone_10.rSet,
                           rDeltaDown := "ЗОНЫ_Параметры".Zone_10.rDeltaDown,
                           rDeltaUp := "ЗОНЫ_Параметры".Zone_10.rDeltaUP,
                           bPriority := "ЗОНЫ_Параметры".Zone_10.bPriority,
                           bInSetpoint => "ЗОНЫ_Параметры".Zone_10.bOUT_ZoneStatus.bInSetpoint,
                           bOutOfRange => "ЗОНЫ_Параметры".Zone_10.bOUT_ZoneStatus.bOutOfRange,
                           bHasPriority => "ЗОНЫ_Параметры".Zone_10.bOUT_ZoneStatus.bHasPriority);
END_REGION

REGION Network 11 (SCL): Соответствие выхода с датчика температур с входом для темп зоны
   "ЗОНЫ_Параметры".Zone_1.rTemp := "AI_DB".AI_1.rAI_Value;
   "ЗОНЫ_Параметры".Zone_2.rTemp := "AI_DB".AI_2.rAI_Value;
   "ЗОНЫ_Параметры".Zone_3.rTemp := "AI_DB".AI_3.rAI_Value;
   "ЗОНЫ_Параметры".Zone_4.rTemp := "AI_DB".AI_4.rAI_Value;
   "ЗОНЫ_Параметры".Zone_5.rTemp := "AI_DB".AI_5.rAI_Value;
   "ЗОНЫ_Параметры".Zone_6.rTemp := "AI_DB".AI_6.rAI_Value;
   "ЗОНЫ_Параметры".Zone_7.rTemp := "AI_DB".AI_7.rAI_Value;
   "ЗОНЫ_Параметры".Zone_8.rTemp := "AI_DB".AI_7.rAI_Value;
   "ЗОНЫ_Параметры".Zone_9.rTemp := "AI_DB".AI_7.rAI_Value;
   "ЗОНЫ_Параметры".Zone_10.rTemp := "AI_DB".AI_7.rAI_Value;
END_REGION
END_FUNCTION

FUNCTION "Аварии/res" : Void   // FC4, LAD
{ S7_Optimized_Access := 'TRUE' }
VERSION : 0.1
   VAR_INPUT
      bResrt : Bool;
   END_VAR
   VAR_OUTPUT
      xAlarm : Bool;   // Есть активные аварии
   END_VAR
BEGIN

REGION Network 1
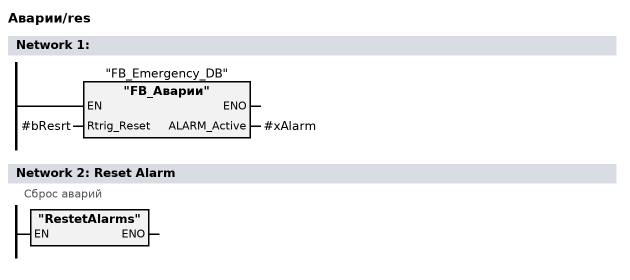
   RUNG wire#powerrail
      "FB_Emergency_DB"(Rtrig_Reset := #bResrt, ALARM_Active => #xAlarm)
   END_RUNG
   // the same network as SCL:
   "FB_Emergency_DB"(Rtrig_Reset := #bResrt, ALARM_Active => #xAlarm);   // "FB_Аварии"
END_REGION

REGION Network 2: Reset Alarm
   // Сброс аварий
   RUNG wire#powerrail
      "RestetAlarms"()
   END_RUNG
   // the same network as SCL:
   "RestetAlarms"();
END_REGION

REGION Network 3 (SCL): Есть активные аварии
END_REGION
END_FUNCTION

FUNCTION "Насосы" : Void   // FC5, LAD
{ S7_Optimized_Access := 'TRUE' }
VERSION : 0.1
// Блоки управления Насосами
BEGIN

REGION Network 1: Насос 1
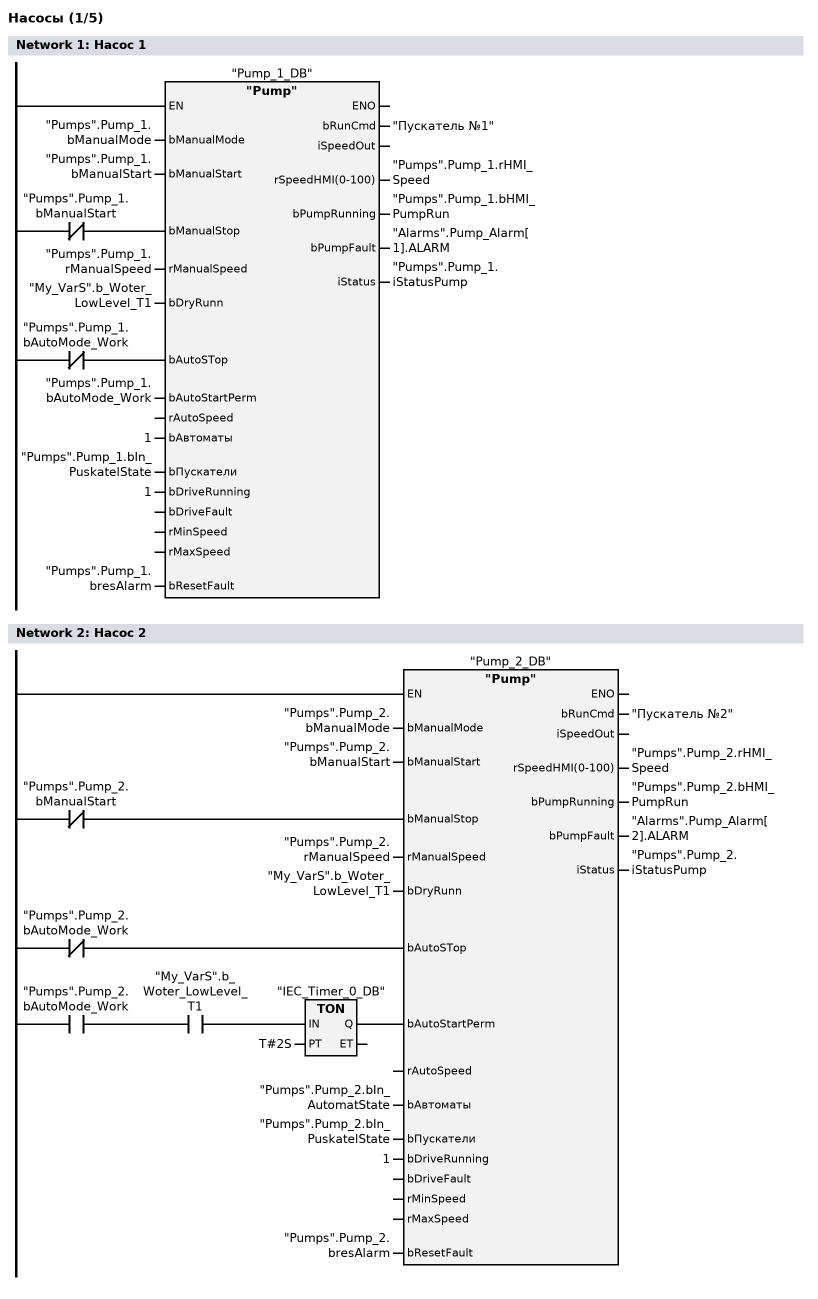
   RUNG wire#powerrail
      "Pump_1_DB"(bManualStop := wire#w1, bAutoSTop := wire#w2, bManualMode := "Pumps".Pump_1.bManualMode, bManualStart := "Pumps".Pump_1.bManualStart, rManualSpeed := "Pumps".Pump_1.rManualSpeed, bDryRunn := "My_VarS".b_Woter_LowLevel_T1, bAutoStartPerm := "Pumps".Pump_1.bAutoMode_Work, rAutoSpeed :=, bАвтоматы := 1, bПускатели := "Pumps".Pump_1.bIn_PuskatelState, bDriveRunning := 1, bDriveFault :=, rMinSpeed :=, rMaxSpeed :=, bResetFault := "Pumps".Pump_1.bresAlarm, bRunCmd => "Пускатель №1", iSpeedOut =>, "rSpeedHMI(0-100)" => "Pumps".Pump_1.rHMI_Speed, bPumpRunning => "Pumps".Pump_1.bHMI_PumpRun, bPumpFault => "Alarms".Pump_Alarm[1].ALARM, iStatus => "Pumps".Pump_1.iStatusPump)
   END_RUNG
   RUNG wire#powerrail
      I_Contact( "Pumps".Pump_1.bManualStart )
   END_RUNG wire#w1
   RUNG wire#powerrail
      I_Contact( "Pumps".Pump_1.bAutoMode_Work )
   END_RUNG wire#w2
   // the same network as SCL:
   "Pump_1_DB"(bManualMode := "Pumps".Pump_1.bManualMode,   // "Pump"
               bManualStart := "Pumps".Pump_1.bManualStart,
               bManualStop := NOT "Pumps".Pump_1.bManualStart,
               rManualSpeed := "Pumps".Pump_1.rManualSpeed,
               bDryRunn := "My_VarS".b_Woter_LowLevel_T1,
               bAutoSTop := NOT "Pumps".Pump_1.bAutoMode_Work,
               bAutoStartPerm := "Pumps".Pump_1.bAutoMode_Work,
               bАвтоматы := 1,
               bПускатели := "Pumps".Pump_1.bIn_PuskatelState,
               bDriveRunning := 1,
               bResetFault := "Pumps".Pump_1.bresAlarm,
               bRunCmd => "Пускатель №1",
               "rSpeedHMI(0-100)" => "Pumps".Pump_1.rHMI_Speed,
               bPumpRunning => "Pumps".Pump_1.bHMI_PumpRun,
               bPumpFault => "Alarms".Pump_Alarm[1].ALARM,
               iStatus => "Pumps".Pump_1.iStatusPump);
END_REGION

REGION Network 2: Насос 2
   "IEC_Timer_0_DB".TON(IN := "Pumps".Pump_2.bAutoMode_Work AND "My_VarS".b_Woter_LowLevel_T1, PT := T#2S);
   "Pump_2_DB"(bManualMode := "Pumps".Pump_2.bManualMode,   // "Pump"
               bManualStart := "Pumps".Pump_2.bManualStart,
               bManualStop := NOT "Pumps".Pump_2.bManualStart,
               rManualSpeed := "Pumps".Pump_2.rManualSpeed,
               bDryRunn := "My_VarS".b_Woter_LowLevel_T1,
               bAutoSTop := NOT "Pumps".Pump_2.bAutoMode_Work,
               bAutoStartPerm := "IEC_Timer_0_DB".Q,
               bАвтоматы := "Pumps".Pump_2.bIn_AutomatState,
               bПускатели := "Pumps".Pump_2.bIn_PuskatelState,
               bDriveRunning := 1,
               bResetFault := "Pumps".Pump_2.bresAlarm,
               bRunCmd => "Пускатель №2",
               "rSpeedHMI(0-100)" => "Pumps".Pump_2.rHMI_Speed,
               bPumpRunning => "Pumps".Pump_2.bHMI_PumpRun,
               bPumpFault => "Alarms".Pump_Alarm[2].ALARM,
               iStatus => "Pumps".Pump_2.iStatusPump);
END_REGION

REGION Network 3: Насос 3
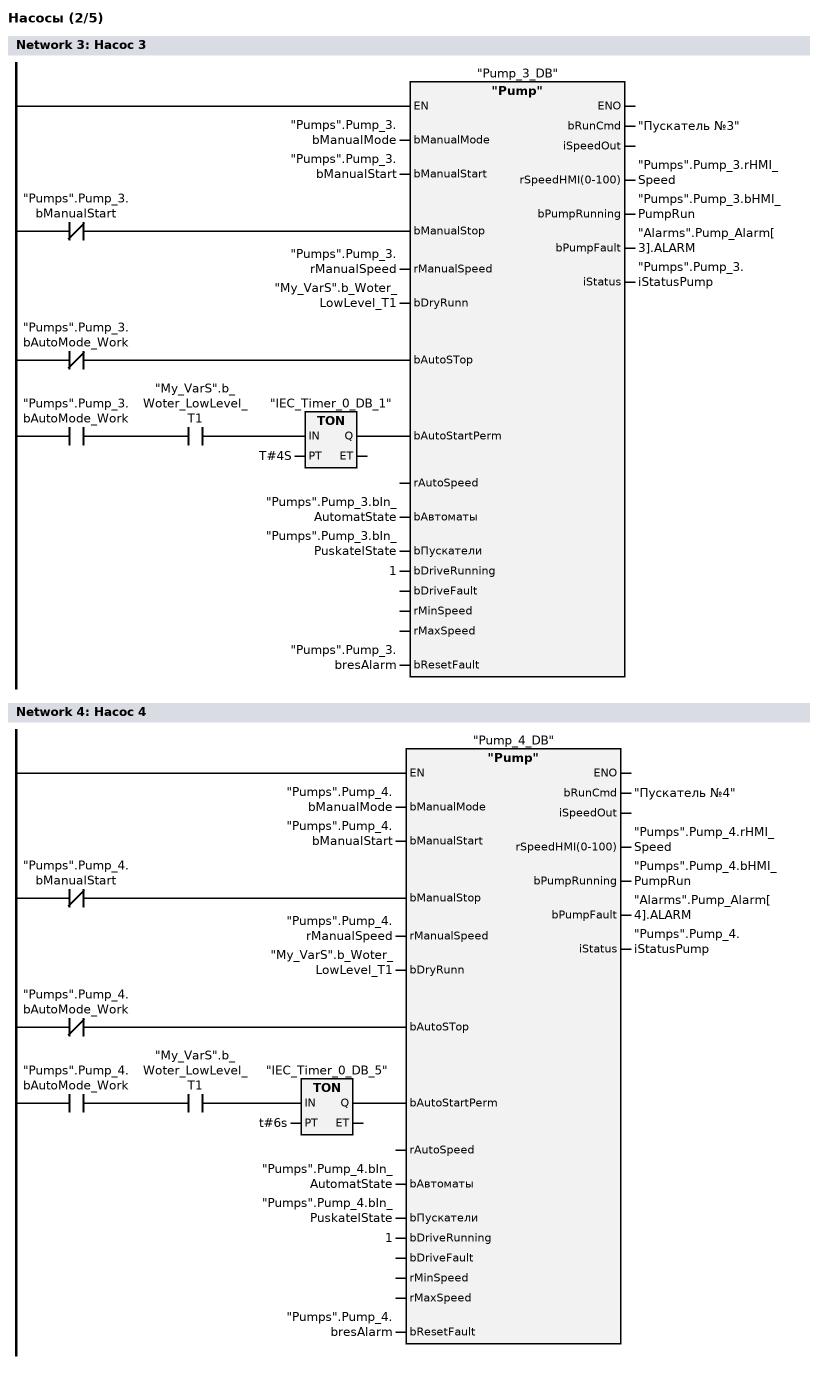
   "IEC_Timer_0_DB_1".TON(IN := "Pumps".Pump_3.bAutoMode_Work AND "My_VarS".b_Woter_LowLevel_T1, PT := T#4S);
   "Pump_3_DB"(bManualMode := "Pumps".Pump_3.bManualMode,   // "Pump"
               bManualStart := "Pumps".Pump_3.bManualStart,
               bManualStop := NOT "Pumps".Pump_3.bManualStart,
               rManualSpeed := "Pumps".Pump_3.rManualSpeed,
               bDryRunn := "My_VarS".b_Woter_LowLevel_T1,
               bAutoSTop := NOT "Pumps".Pump_3.bAutoMode_Work,
               bAutoStartPerm := "IEC_Timer_0_DB_1".Q,
               bАвтоматы := "Pumps".Pump_3.bIn_AutomatState,
               bПускатели := "Pumps".Pump_3.bIn_PuskatelState,
               bDriveRunning := 1,
               bResetFault := "Pumps".Pump_3.bresAlarm,
               bRunCmd => "Пускатель №3",
               "rSpeedHMI(0-100)" => "Pumps".Pump_3.rHMI_Speed,
               bPumpRunning => "Pumps".Pump_3.bHMI_PumpRun,
               bPumpFault => "Alarms".Pump_Alarm[3].ALARM,
               iStatus => "Pumps".Pump_3.iStatusPump);
END_REGION

REGION Network 4: Насос 4
   "IEC_Timer_0_DB_5".TON(IN := "Pumps".Pump_4.bAutoMode_Work AND "My_VarS".b_Woter_LowLevel_T1, PT := t#6s);
   "Pump_4_DB"(bManualMode := "Pumps".Pump_4.bManualMode,   // "Pump"
               bManualStart := "Pumps".Pump_4.bManualStart,
               bManualStop := NOT "Pumps".Pump_4.bManualStart,
               rManualSpeed := "Pumps".Pump_4.rManualSpeed,
               bDryRunn := "My_VarS".b_Woter_LowLevel_T1,
               bAutoSTop := NOT "Pumps".Pump_4.bAutoMode_Work,
               bAutoStartPerm := "IEC_Timer_0_DB_5".Q,
               bАвтоматы := "Pumps".Pump_4.bIn_AutomatState,
               bПускатели := "Pumps".Pump_4.bIn_PuskatelState,
               bDriveRunning := 1,
               bResetFault := "Pumps".Pump_4.bresAlarm,
               bRunCmd => "Пускатель №4",
               "rSpeedHMI(0-100)" => "Pumps".Pump_4.rHMI_Speed,
               bPumpRunning => "Pumps".Pump_4.bHMI_PumpRun,
               bPumpFault => "Alarms".Pump_Alarm[4].ALARM,
               iStatus => "Pumps".Pump_4.iStatusPump);
END_REGION

REGION Network 5: Насос 5
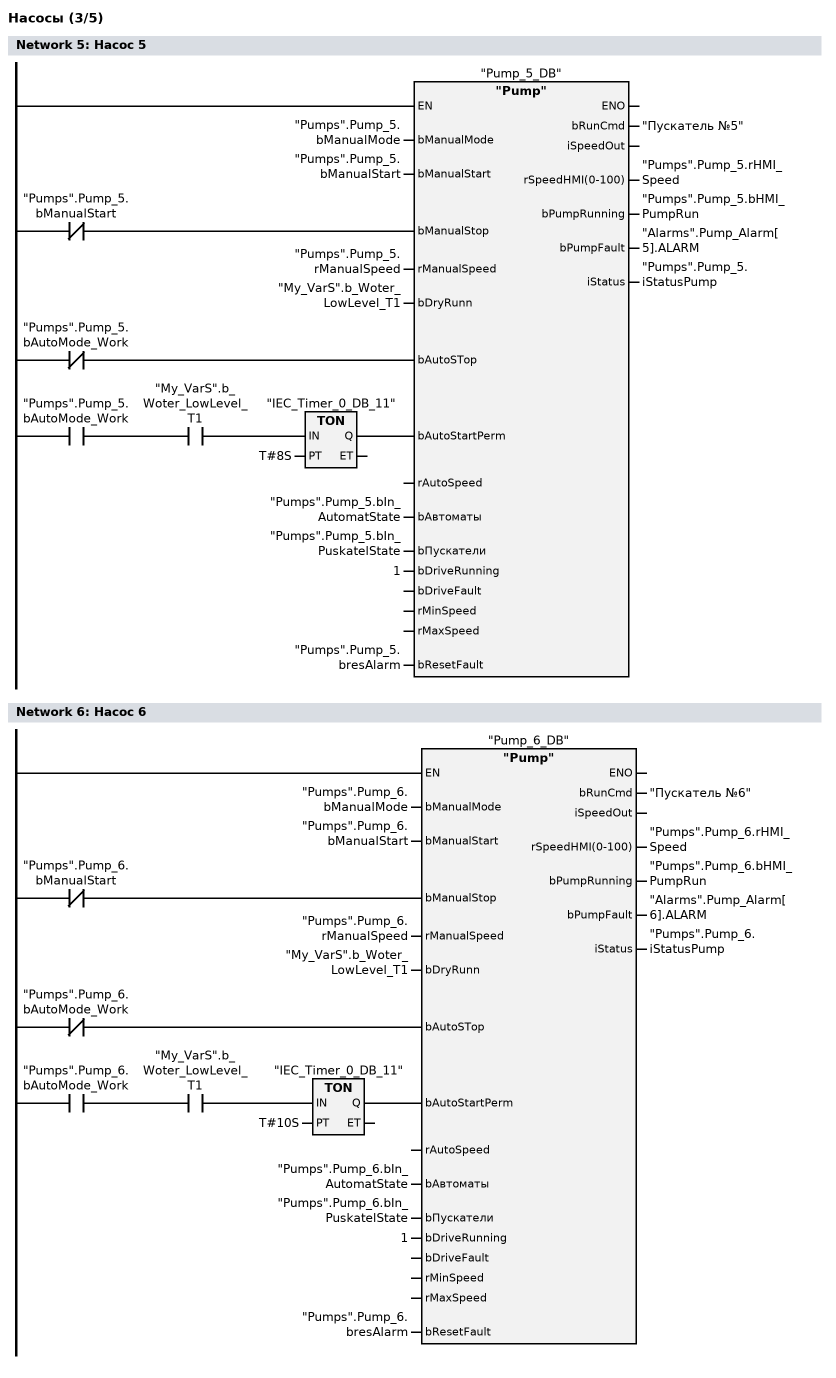
   "IEC_Timer_0_DB_11".TON(IN := "Pumps".Pump_5.bAutoMode_Work AND "My_VarS".b_Woter_LowLevel_T1, PT := T#8S);
   "Pump_5_DB"(bManualMode := "Pumps".Pump_5.bManualMode,   // "Pump"
               bManualStart := "Pumps".Pump_5.bManualStart,
               bManualStop := NOT "Pumps".Pump_5.bManualStart,
               rManualSpeed := "Pumps".Pump_5.rManualSpeed,
               bDryRunn := "My_VarS".b_Woter_LowLevel_T1,
               bAutoSTop := NOT "Pumps".Pump_5.bAutoMode_Work,
               bAutoStartPerm := "IEC_Timer_0_DB_11".Q,
               bАвтоматы := "Pumps".Pump_5.bIn_AutomatState,
               bПускатели := "Pumps".Pump_5.bIn_PuskatelState,
               bDriveRunning := 1,
               bResetFault := "Pumps".Pump_5.bresAlarm,
               bRunCmd => "Пускатель №5",
               "rSpeedHMI(0-100)" => "Pumps".Pump_5.rHMI_Speed,
               bPumpRunning => "Pumps".Pump_5.bHMI_PumpRun,
               bPumpFault => "Alarms".Pump_Alarm[5].ALARM,
               iStatus => "Pumps".Pump_5.iStatusPump);
END_REGION

REGION Network 6: Насос 6
   "IEC_Timer_0_DB_11".TON(IN := "Pumps".Pump_6.bAutoMode_Work AND "My_VarS".b_Woter_LowLevel_T1, PT := T#10S);
   "Pump_6_DB"(bManualMode := "Pumps".Pump_6.bManualMode,   // "Pump"
               bManualStart := "Pumps".Pump_6.bManualStart,
               bManualStop := NOT "Pumps".Pump_6.bManualStart,
               rManualSpeed := "Pumps".Pump_6.rManualSpeed,
               bDryRunn := "My_VarS".b_Woter_LowLevel_T1,
               bAutoSTop := NOT "Pumps".Pump_6.bAutoMode_Work,
               bAutoStartPerm := "IEC_Timer_0_DB_11".Q,
               bАвтоматы := "Pumps".Pump_6.bIn_AutomatState,
               bПускатели := "Pumps".Pump_6.bIn_PuskatelState,
               bDriveRunning := 1,
               bResetFault := "Pumps".Pump_6.bresAlarm,
               bRunCmd => "Пускатель №6",
               "rSpeedHMI(0-100)" => "Pumps".Pump_6.rHMI_Speed,
               bPumpRunning => "Pumps".Pump_6.bHMI_PumpRun,
               bPumpFault => "Alarms".Pump_Alarm[6].ALARM,
               iStatus => "Pumps".Pump_6.iStatusPump);
END_REGION

REGION Network 7: Насос 7
   // Задержка на выключение для насоса по холоду, что бы не примерзло ничего ждем когда клапан закроется - потом выключаем насос
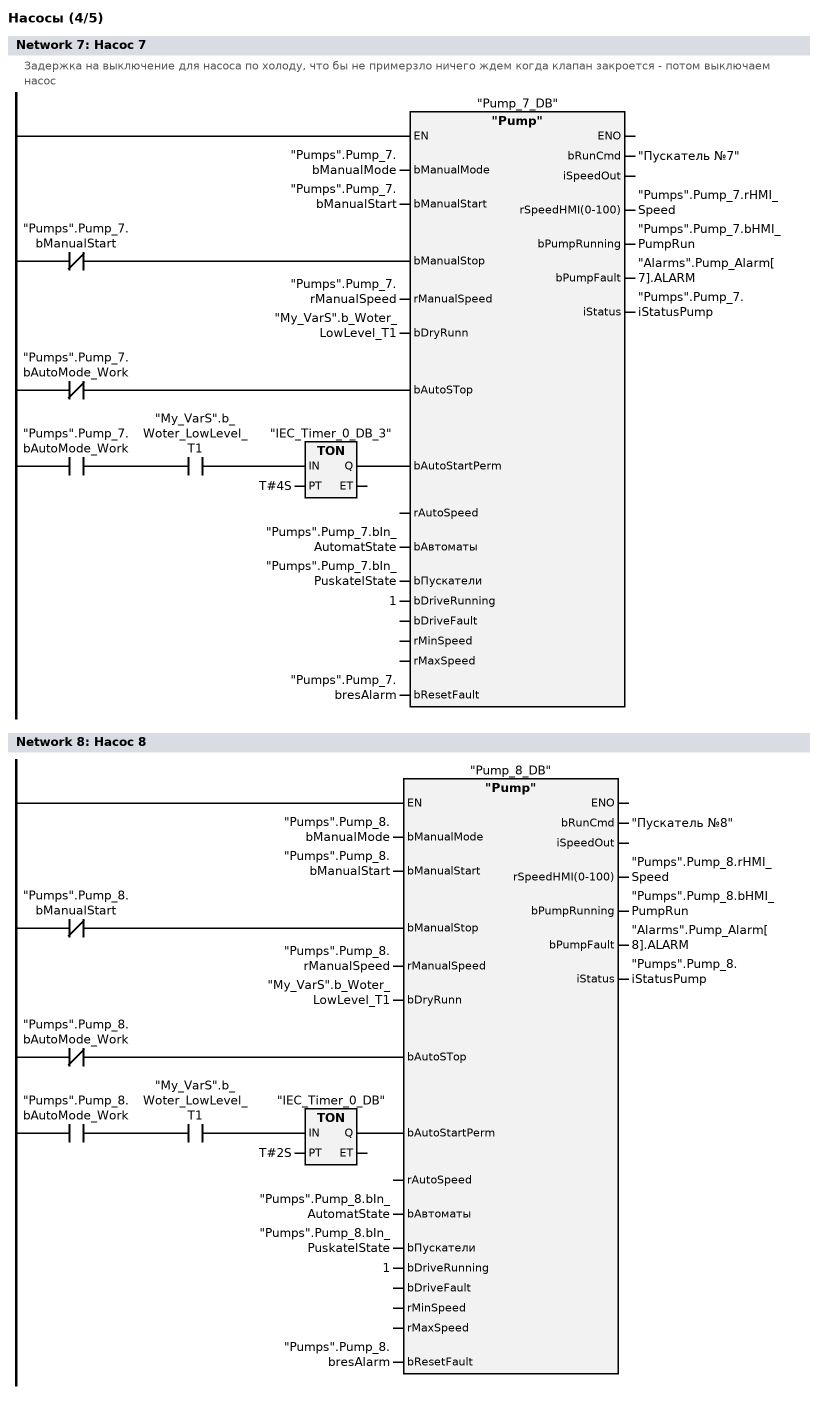
   "IEC_Timer_0_DB_3".TON(IN := "Pumps".Pump_7.bAutoMode_Work AND "My_VarS".b_Woter_LowLevel_T1, PT := T#4S);
   "Pump_7_DB"(bManualMode := "Pumps".Pump_7.bManualMode,   // "Pump"
               bManualStart := "Pumps".Pump_7.bManualStart,
               bManualStop := NOT "Pumps".Pump_7.bManualStart,
               rManualSpeed := "Pumps".Pump_7.rManualSpeed,
               bDryRunn := "My_VarS".b_Woter_LowLevel_T1,
               bAutoSTop := NOT "Pumps".Pump_7.bAutoMode_Work,
               bAutoStartPerm := "IEC_Timer_0_DB_3".Q,
               bАвтоматы := "Pumps".Pump_7.bIn_AutomatState,
               bПускатели := "Pumps".Pump_7.bIn_PuskatelState,
               bDriveRunning := 1,
               bResetFault := "Pumps".Pump_7.bresAlarm,
               bRunCmd => "Пускатель №7",
               "rSpeedHMI(0-100)" => "Pumps".Pump_7.rHMI_Speed,
               bPumpRunning => "Pumps".Pump_7.bHMI_PumpRun,
               bPumpFault => "Alarms".Pump_Alarm[7].ALARM,
               iStatus => "Pumps".Pump_7.iStatusPump);
END_REGION

REGION Network 8: Насос 8
   "IEC_Timer_0_DB".TON(IN := "Pumps".Pump_8.bAutoMode_Work AND "My_VarS".b_Woter_LowLevel_T1, PT := T#2S);
   "Pump_8_DB"(bManualMode := "Pumps".Pump_8.bManualMode,   // "Pump"
               bManualStart := "Pumps".Pump_8.bManualStart,
               bManualStop := NOT "Pumps".Pump_8.bManualStart,
               rManualSpeed := "Pumps".Pump_8.rManualSpeed,
               bDryRunn := "My_VarS".b_Woter_LowLevel_T1,
               bAutoSTop := NOT "Pumps".Pump_8.bAutoMode_Work,
               bAutoStartPerm := "IEC_Timer_0_DB".Q,
               bАвтоматы := "Pumps".Pump_8.bIn_AutomatState,
               bПускатели := "Pumps".Pump_8.bIn_PuskatelState,
               bDriveRunning := 1,
               bResetFault := "Pumps".Pump_8.bresAlarm,
               bRunCmd => "Пускатель №8",
               "rSpeedHMI(0-100)" => "Pumps".Pump_8.rHMI_Speed,
               bPumpRunning => "Pumps".Pump_8.bHMI_PumpRun,
               bPumpFault => "Alarms".Pump_Alarm[8].ALARM,
               iStatus => "Pumps".Pump_8.iStatusPump);
END_REGION

REGION Network 9: Насос 9
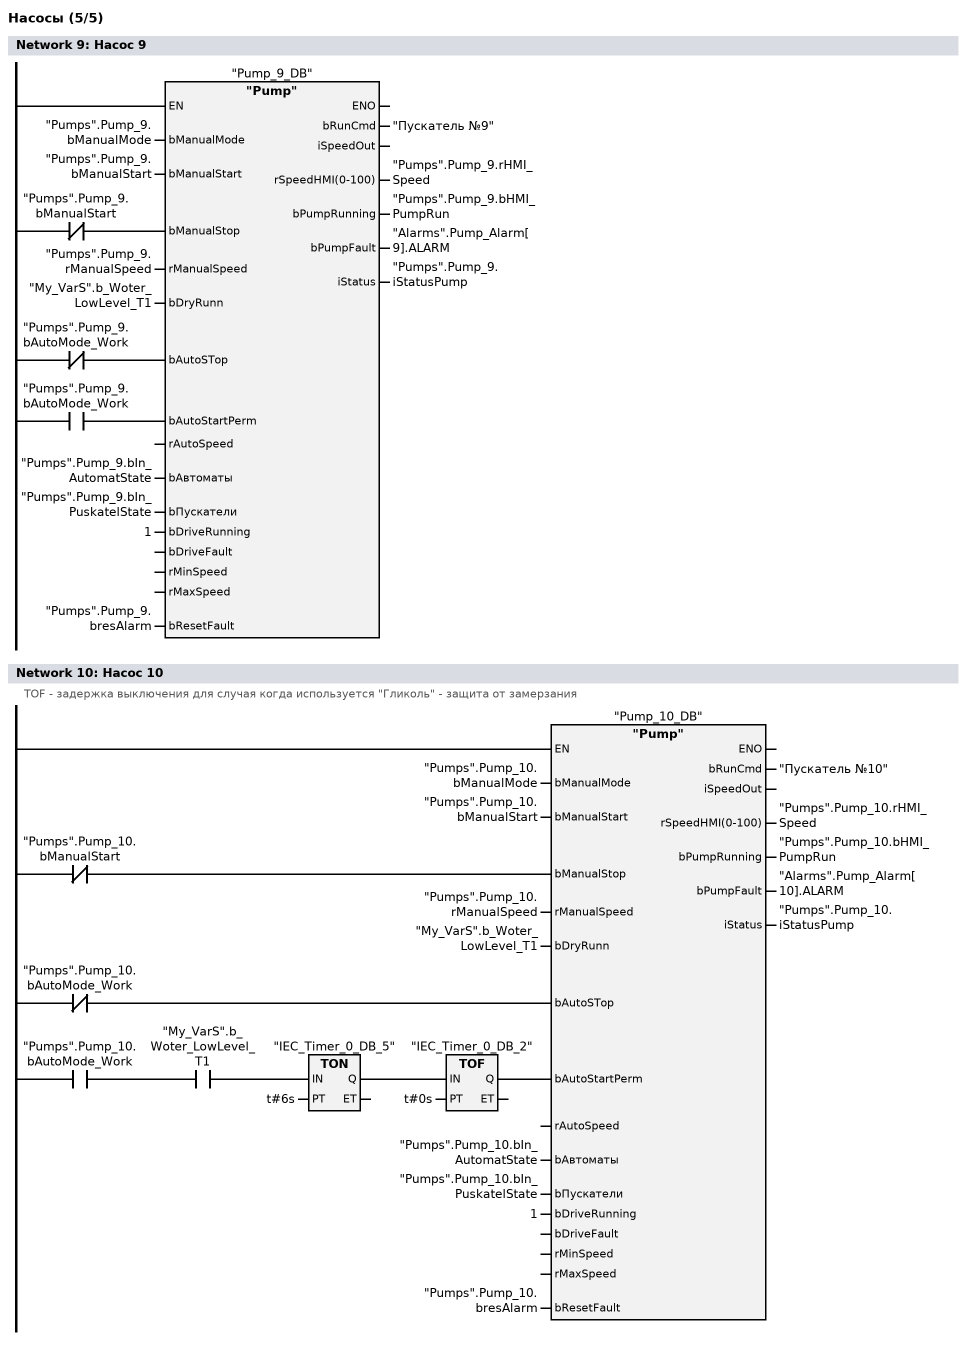
   RUNG wire#powerrail
      "Pump_9_DB"(bManualStop := wire#w1, bAutoSTop := wire#w2, bAutoStartPerm := wire#w3, bManualMode := "Pumps".Pump_9.bManualMode, bManualStart := "Pumps".Pump_9.bManualStart, rManualSpeed := "Pumps".Pump_9.rManualSpeed, bDryRunn := "My_VarS".b_Woter_LowLevel_T1, rAutoSpeed :=, bАвтоматы := "Pumps".Pump_9.bIn_AutomatState, bПускатели := "Pumps".Pump_9.bIn_PuskatelState, bDriveRunning := 1, bDriveFault :=, rMinSpeed :=, rMaxSpeed :=, bResetFault := "Pumps".Pump_9.bresAlarm, bRunCmd => "Пускатель №9", iSpeedOut =>, "rSpeedHMI(0-100)" => "Pumps".Pump_9.rHMI_Speed, bPumpRunning => "Pumps".Pump_9.bHMI_PumpRun, bPumpFault => "Alarms".Pump_Alarm[9].ALARM, iStatus => "Pumps".Pump_9.iStatusPump)
   END_RUNG
   RUNG wire#powerrail
      I_Contact( "Pumps".Pump_9.bManualStart )
   END_RUNG wire#w1
   RUNG wire#powerrail
      I_Contact( "Pumps".Pump_9.bAutoMode_Work )
   END_RUNG wire#w2
   RUNG wire#powerrail
      Contact( "Pumps".Pump_9.bAutoMode_Work )
   END_RUNG wire#w3
   // the same network as SCL:
   "Pump_9_DB"(bManualMode := "Pumps".Pump_9.bManualMode,   // "Pump"
               bManualStart := "Pumps".Pump_9.bManualStart,
               bManualStop := NOT "Pumps".Pump_9.bManualStart,
               rManualSpeed := "Pumps".Pump_9.rManualSpeed,
               bDryRunn := "My_VarS".b_Woter_LowLevel_T1,
               bAutoSTop := NOT "Pumps".Pump_9.bAutoMode_Work,
               bAutoStartPerm := "Pumps".Pump_9.bAutoMode_Work,
               bАвтоматы := "Pumps".Pump_9.bIn_AutomatState,
               bПускатели := "Pumps".Pump_9.bIn_PuskatelState,
               bDriveRunning := 1,
               bResetFault := "Pumps".Pump_9.bresAlarm,
               bRunCmd => "Пускатель №9",
               "rSpeedHMI(0-100)" => "Pumps".Pump_9.rHMI_Speed,
               bPumpRunning => "Pumps".Pump_9.bHMI_PumpRun,
               bPumpFault => "Alarms".Pump_Alarm[9].ALARM,
               iStatus => "Pumps".Pump_9.iStatusPump);
END_REGION

REGION Network 10: Насос 10
   // TOF - задержка выключения для случая когда используется "Гликоль" - защита от замерзания
   "IEC_Timer_0_DB_5".TON(IN := "Pumps".Pump_10.bAutoMode_Work AND "My_VarS".b_Woter_LowLevel_T1, PT := t#6s);
   "IEC_Timer_0_DB_2".TOF(IN := "IEC_Timer_0_DB_5".Q, PT := t#0s);
   "Pump_10_DB"(bManualMode := "Pumps".Pump_10.bManualMode,   // "Pump"
                bManualStart := "Pumps".Pump_10.bManualStart,
                bManualStop := NOT "Pumps".Pump_10.bManualStart,
                rManualSpeed := "Pumps".Pump_10.rManualSpeed,
                bDryRunn := "My_VarS".b_Woter_LowLevel_T1,
                bAutoSTop := NOT "Pumps".Pump_10.bAutoMode_Work,
                bAutoStartPerm := "IEC_Timer_0_DB_2".Q,
                bАвтоматы := "Pumps".Pump_10.bIn_AutomatState,
                bПускатели := "Pumps".Pump_10.bIn_PuskatelState,
                bDriveRunning := 1,
                bResetFault := "Pumps".Pump_10.bresAlarm,
                bRunCmd => "Пускатель №10",
                "rSpeedHMI(0-100)" => "Pumps".Pump_10.rHMI_Speed,
                bPumpRunning => "Pumps".Pump_10.bHMI_PumpRun,
                bPumpFault => "Alarms".Pump_Alarm[10].ALARM,
                iStatus => "Pumps".Pump_10.iStatusPump);
END_REGION
END_FUNCTION

FUNCTION "Analogs_IN_All" : Void   // FC6, LAD
TITLE = Датчики AI
{ S7_Optimized_Access := 'FALSE' }
VERSION : 0.1
// Темп - PT100 - 7 шт
// Давление 4-20 - 0
//  шт
BEGIN

REGION Network 1: Датчик температуры - 1
   // РТ-100
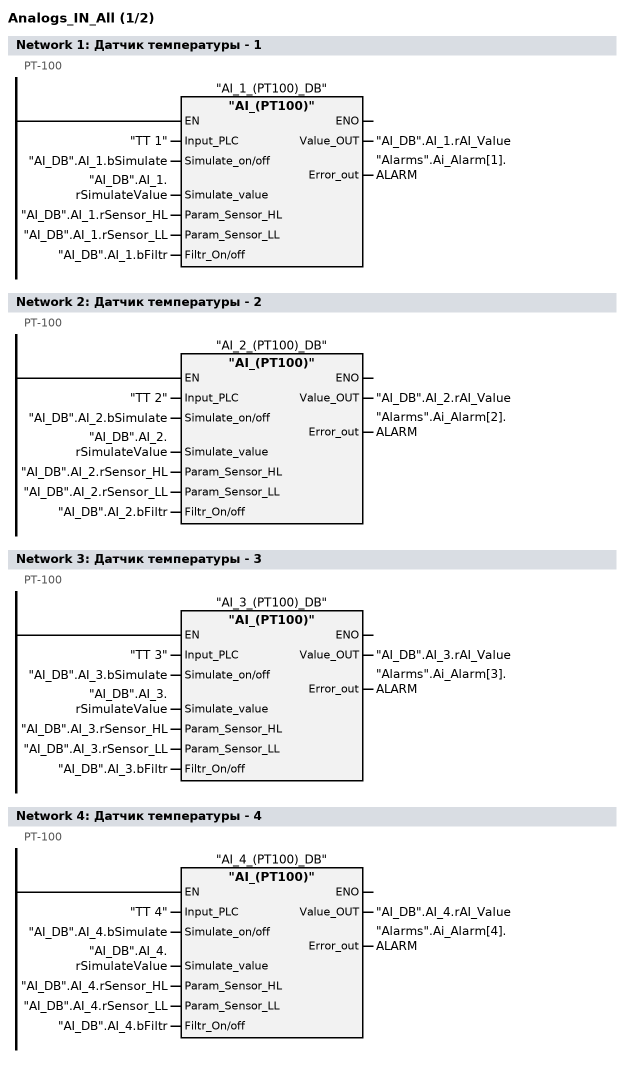
   RUNG wire#powerrail
      "AI_1_(PT100)_DB"(Input_PLC := "TT 1", "Simulate_on/off" := "AI_DB".AI_1.bSimulate, Simulate_value := "AI_DB".AI_1.rSimulateValue, Param_Sensor_HL := "AI_DB".AI_1.rSensor_HL, Param_Sensor_LL := "AI_DB".AI_1.rSensor_LL, "Filtr_On/off" := "AI_DB".AI_1.bFiltr, Value_OUT => "AI_DB".AI_1.rAI_Value, Error_out => "Alarms".Ai_Alarm[1].ALARM)
   END_RUNG
   // the same network as SCL:
   "AI_1_(PT100)_DB"(Input_PLC := "TT 1",   // "AI_(PT100)"
                     "Simulate_on/off" := "AI_DB".AI_1.bSimulate,
                     Simulate_value := "AI_DB".AI_1.rSimulateValue,
                     Param_Sensor_HL := "AI_DB".AI_1.rSensor_HL,
                     Param_Sensor_LL := "AI_DB".AI_1.rSensor_LL,
                     "Filtr_On/off" := "AI_DB".AI_1.bFiltr,
                     Value_OUT => "AI_DB".AI_1.rAI_Value,
                     Error_out => "Alarms".Ai_Alarm[1].ALARM);
END_REGION

REGION Network 2: Датчик температуры - 2
   // РТ-100
   RUNG wire#powerrail
      "AI_2_(PT100)_DB"(Input_PLC := "TT 2", "Simulate_on/off" := "AI_DB".AI_2.bSimulate, Simulate_value := "AI_DB".AI_2.rSimulateValue, Param_Sensor_HL := "AI_DB".AI_2.rSensor_HL, Param_Sensor_LL := "AI_DB".AI_2.rSensor_LL, "Filtr_On/off" := "AI_DB".AI_2.bFiltr, Value_OUT => "AI_DB".AI_2.rAI_Value, Error_out => "Alarms".Ai_Alarm[2].ALARM)
   END_RUNG
   // the same network as SCL:
   "AI_2_(PT100)_DB"(Input_PLC := "TT 2",   // "AI_(PT100)"
                     "Simulate_on/off" := "AI_DB".AI_2.bSimulate,
                     Simulate_value := "AI_DB".AI_2.rSimulateValue,
                     Param_Sensor_HL := "AI_DB".AI_2.rSensor_HL,
                     Param_Sensor_LL := "AI_DB".AI_2.rSensor_LL,
                     "Filtr_On/off" := "AI_DB".AI_2.bFiltr,
                     Value_OUT => "AI_DB".AI_2.rAI_Value,
                     Error_out => "Alarms".Ai_Alarm[2].ALARM);
END_REGION

REGION Network 3: Датчик температуры - 3
   // РТ-100
   RUNG wire#powerrail
      "AI_3_(PT100)_DB"(Input_PLC := "TT 3", "Simulate_on/off" := "AI_DB".AI_3.bSimulate, Simulate_value := "AI_DB".AI_3.rSimulateValue, Param_Sensor_HL := "AI_DB".AI_3.rSensor_HL, Param_Sensor_LL := "AI_DB".AI_3.rSensor_LL, "Filtr_On/off" := "AI_DB".AI_3.bFiltr, Value_OUT => "AI_DB".AI_3.rAI_Value, Error_out => "Alarms".Ai_Alarm[3].ALARM)
   END_RUNG
   // the same network as SCL:
   "AI_3_(PT100)_DB"(Input_PLC := "TT 3",   // "AI_(PT100)"
                     "Simulate_on/off" := "AI_DB".AI_3.bSimulate,
                     Simulate_value := "AI_DB".AI_3.rSimulateValue,
                     Param_Sensor_HL := "AI_DB".AI_3.rSensor_HL,
                     Param_Sensor_LL := "AI_DB".AI_3.rSensor_LL,
                     "Filtr_On/off" := "AI_DB".AI_3.bFiltr,
                     Value_OUT => "AI_DB".AI_3.rAI_Value,
                     Error_out => "Alarms".Ai_Alarm[3].ALARM);
END_REGION

REGION Network 4: Датчик температуры - 4
   // РТ-100
   RUNG wire#powerrail
      "AI_4_(PT100)_DB"(Input_PLC := "TT 4", "Simulate_on/off" := "AI_DB".AI_4.bSimulate, Simulate_value := "AI_DB".AI_4.rSimulateValue, Param_Sensor_HL := "AI_DB".AI_4.rSensor_HL, Param_Sensor_LL := "AI_DB".AI_4.rSensor_LL, "Filtr_On/off" := "AI_DB".AI_4.bFiltr, Value_OUT => "AI_DB".AI_4.rAI_Value, Error_out => "Alarms".Ai_Alarm[4].ALARM)
   END_RUNG
   // the same network as SCL:
   "AI_4_(PT100)_DB"(Input_PLC := "TT 4",   // "AI_(PT100)"
                     "Simulate_on/off" := "AI_DB".AI_4.bSimulate,
                     Simulate_value := "AI_DB".AI_4.rSimulateValue,
                     Param_Sensor_HL := "AI_DB".AI_4.rSensor_HL,
                     Param_Sensor_LL := "AI_DB".AI_4.rSensor_LL,
                     "Filtr_On/off" := "AI_DB".AI_4.bFiltr,
                     Value_OUT => "AI_DB".AI_4.rAI_Value,
                     Error_out => "Alarms".Ai_Alarm[4].ALARM);
END_REGION

REGION Network 5: Датчик температуры - 5
   // РТ-100
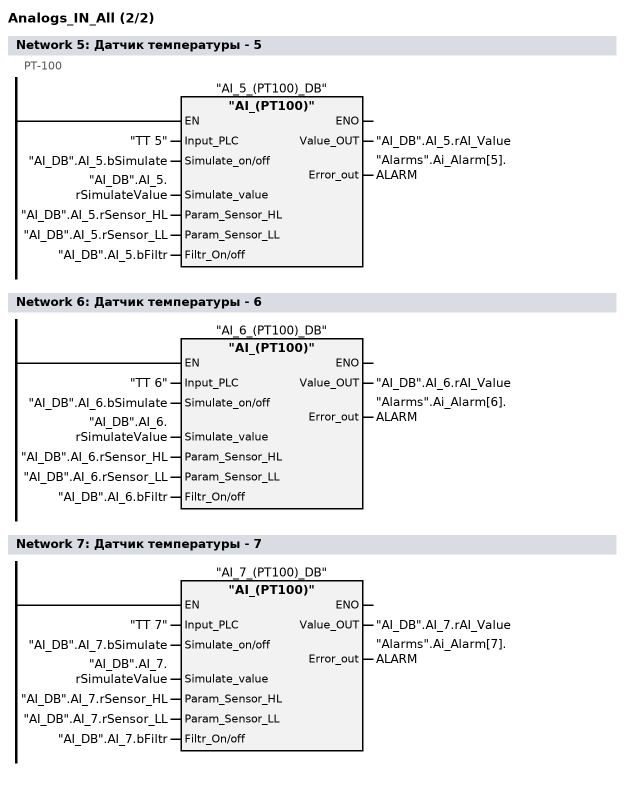
   RUNG wire#powerrail
      "AI_5_(PT100)_DB"(Input_PLC := "TT 5", "Simulate_on/off" := "AI_DB".AI_5.bSimulate, Simulate_value := "AI_DB".AI_5.rSimulateValue, Param_Sensor_HL := "AI_DB".AI_5.rSensor_HL, Param_Sensor_LL := "AI_DB".AI_5.rSensor_LL, "Filtr_On/off" := "AI_DB".AI_5.bFiltr, Value_OUT => "AI_DB".AI_5.rAI_Value, Error_out => "Alarms".Ai_Alarm[5].ALARM)
   END_RUNG
   // the same network as SCL:
   "AI_5_(PT100)_DB"(Input_PLC := "TT 5",   // "AI_(PT100)"
                     "Simulate_on/off" := "AI_DB".AI_5.bSimulate,
                     Simulate_value := "AI_DB".AI_5.rSimulateValue,
                     Param_Sensor_HL := "AI_DB".AI_5.rSensor_HL,
                     Param_Sensor_LL := "AI_DB".AI_5.rSensor_LL,
                     "Filtr_On/off" := "AI_DB".AI_5.bFiltr,
                     Value_OUT => "AI_DB".AI_5.rAI_Value,
                     Error_out => "Alarms".Ai_Alarm[5].ALARM);
END_REGION

REGION Network 6: Датчик температуры - 6
   RUNG wire#powerrail
      "AI_6_(PT100)_DB"(Input_PLC := "TT 6", "Simulate_on/off" := "AI_DB".AI_6.bSimulate, Simulate_value := "AI_DB".AI_6.rSimulateValue, Param_Sensor_HL := "AI_DB".AI_6.rSensor_HL, Param_Sensor_LL := "AI_DB".AI_6.rSensor_LL, "Filtr_On/off" := "AI_DB".AI_6.bFiltr, Value_OUT => "AI_DB".AI_6.rAI_Value, Error_out => "Alarms".Ai_Alarm[6].ALARM)
   END_RUNG
   // the same network as SCL:
   "AI_6_(PT100)_DB"(Input_PLC := "TT 6",   // "AI_(PT100)"
                     "Simulate_on/off" := "AI_DB".AI_6.bSimulate,
                     Simulate_value := "AI_DB".AI_6.rSimulateValue,
                     Param_Sensor_HL := "AI_DB".AI_6.rSensor_HL,
                     Param_Sensor_LL := "AI_DB".AI_6.rSensor_LL,
                     "Filtr_On/off" := "AI_DB".AI_6.bFiltr,
                     Value_OUT => "AI_DB".AI_6.rAI_Value,
                     Error_out => "Alarms".Ai_Alarm[6].ALARM);
END_REGION

REGION Network 7: Датчик температуры - 7
   RUNG wire#powerrail
      "AI_7_(PT100)_DB"(Input_PLC := "TT 7", "Simulate_on/off" := "AI_DB".AI_7.bSimulate, Simulate_value := "AI_DB".AI_7.rSimulateValue, Param_Sensor_HL := "AI_DB".AI_7.rSensor_HL, Param_Sensor_LL := "AI_DB".AI_7.rSensor_LL, "Filtr_On/off" := "AI_DB".AI_7.bFiltr, Value_OUT => "AI_DB".AI_7.rAI_Value, Error_out => "Alarms".Ai_Alarm[7].ALARM)
   END_RUNG
   // the same network as SCL:
   "AI_7_(PT100)_DB"(Input_PLC := "TT 7",   // "AI_(PT100)"
                     "Simulate_on/off" := "AI_DB".AI_7.bSimulate,
                     Simulate_value := "AI_DB".AI_7.rSimulateValue,
                     Param_Sensor_HL := "AI_DB".AI_7.rSensor_HL,
                     Param_Sensor_LL := "AI_DB".AI_7.rSensor_LL,
                     "Filtr_On/off" := "AI_DB".AI_7.bFiltr,
                     Value_OUT => "AI_DB".AI_7.rAI_Value,
                     Error_out => "Alarms".Ai_Alarm[7].ALARM);
END_REGION
END_FUNCTION

FUNCTION "Discret_Inputs_All" : Void   // FC8, LAD
TITLE = Для сбора всех DI в одном месте
{ S7_Optimized_Access := 'FALSE' }
VERSION : 0.1
   VAR CONSTANT
      Cons_TimeDelay : DInt := 100;
   END_VAR
BEGIN

REGION Network 1: E-Stop1
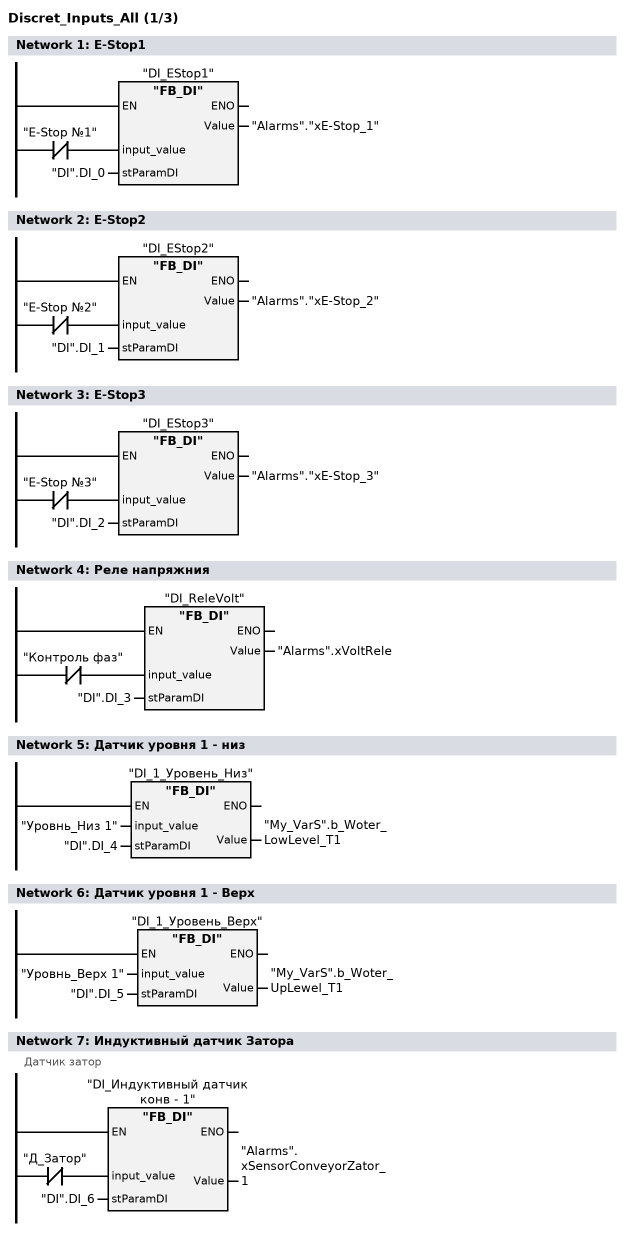
   RUNG wire#powerrail
      "DI_EStop1"(input_value := wire#w1, stParamDI := "DI".DI_0, Value => "Alarms"."xE-Stop_1")
   END_RUNG
   RUNG wire#powerrail
      I_Contact( "E-Stop №1" )
   END_RUNG wire#w1
   // the same network as SCL:
   "DI_EStop1"(input_value := NOT "E-Stop №1", stParamDI := "DI".DI_0, Value => "Alarms"."xE-Stop_1");   // "FB_DI"
END_REGION

REGION Network 2: E-Stop2
   RUNG wire#powerrail
      "DI_EStop2"(input_value := wire#w1, stParamDI := "DI".DI_1, Value => "Alarms"."xE-Stop_2")
   END_RUNG
   RUNG wire#powerrail
      I_Contact( "E-Stop №2" )
   END_RUNG wire#w1
   // the same network as SCL:
   "DI_EStop2"(input_value := NOT "E-Stop №2", stParamDI := "DI".DI_1, Value => "Alarms"."xE-Stop_2");   // "FB_DI"
END_REGION

REGION Network 3: E-Stop3
   RUNG wire#powerrail
      "DI_EStop3"(input_value := wire#w1, stParamDI := "DI".DI_2, Value => "Alarms"."xE-Stop_3")
   END_RUNG
   RUNG wire#powerrail
      I_Contact( "E-Stop №3" )
   END_RUNG wire#w1
   // the same network as SCL:
   "DI_EStop3"(input_value := NOT "E-Stop №3", stParamDI := "DI".DI_2, Value => "Alarms"."xE-Stop_3");   // "FB_DI"
END_REGION

REGION Network 4: Реле напряжния
   RUNG wire#powerrail
      "DI_ReleVolt"(input_value := wire#w1, stParamDI := "DI".DI_3, Value => "Alarms".xVoltRele)
   END_RUNG
   RUNG wire#powerrail
      I_Contact( "Контроль фаз" )
   END_RUNG wire#w1
   // the same network as SCL:
   "DI_ReleVolt"(input_value := NOT "Контроль фаз", stParamDI := "DI".DI_3, Value => "Alarms".xVoltRele);   // "FB_DI"
END_REGION

REGION Network 5: Датчик уровня 1 - низ
   RUNG wire#powerrail
      "DI_1_Уровень_Низ"(input_value := "Уровнь_Низ 1", stParamDI := "DI".DI_4, Value => "My_VarS".b_Woter_LowLevel_T1)
   END_RUNG
   // the same network as SCL:
   "DI_1_Уровень_Низ"(input_value := "Уровнь_Низ 1",   // "FB_DI"
                      stParamDI := "DI".DI_4,
                      Value => "My_VarS".b_Woter_LowLevel_T1);
END_REGION

REGION Network 6: Датчик уровня 1 - Верх
   RUNG wire#powerrail
      "DI_1_Уровень_Верх"(input_value := "Уровнь_Верх 1", stParamDI := "DI".DI_5, Value => "My_VarS".b_Woter_UpLewel_T1)
   END_RUNG
   // the same network as SCL:
   "DI_1_Уровень_Верх"(input_value := "Уровнь_Верх 1",   // "FB_DI"
                       stParamDI := "DI".DI_5,
                       Value => "My_VarS".b_Woter_UpLewel_T1);
END_REGION

REGION Network 7: Индуктивный датчик Затора
   // Датчик затор
   RUNG wire#powerrail
      "DI_Индуктивный датчик конв - 1"(input_value := wire#w1, stParamDI := "DI".DI_6, Value => "Alarms".xSensorConveyorZator_1)
   END_RUNG
   RUNG wire#powerrail
      I_Contact( "Д_Затор" )
   END_RUNG wire#w1
   // the same network as SCL:
   "DI_Индуктивный датчик конв - 1"(input_value := NOT "Д_Затор",   // "FB_DI"
                           stParamDI := "DI".DI_6,
                           Value => "Alarms".xSensorConveyorZator_1);
END_REGION

REGION Network 8: Работа чатотника - 1
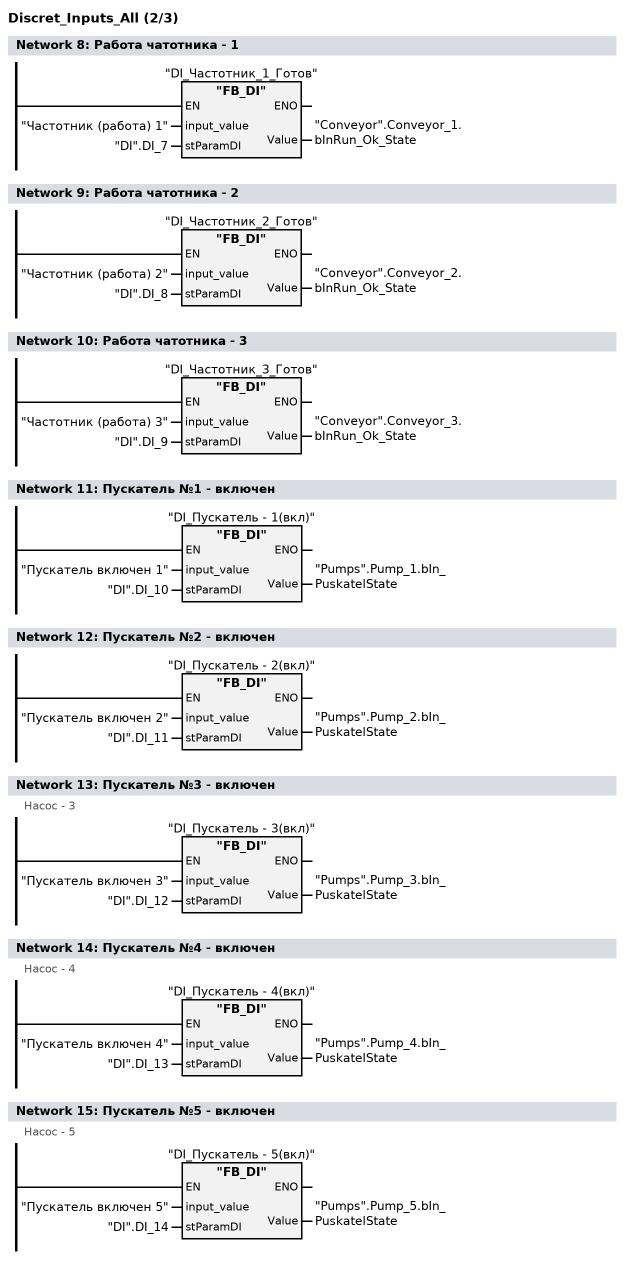
   RUNG wire#powerrail
      "DI_Частотник_1_Готов"(input_value := "Частотник (работа) 1", stParamDI := "DI".DI_7, Value => "Conveyor".Conveyor_1.bInRun_Ok_State)
   END_RUNG
   // the same network as SCL:
   "DI_Частотник_1_Готов"(input_value := "Частотник (работа) 1",   // "FB_DI"
                          stParamDI := "DI".DI_7,
                          Value => "Conveyor".Conveyor_1.bInRun_Ok_State);
END_REGION

REGION Network 9: Работа чатотника - 2
   RUNG wire#powerrail
      "DI_Частотник_2_Готов"(input_value := "Частотник (работа) 2", stParamDI := "DI".DI_8, Value => "Conveyor".Conveyor_2.bInRun_Ok_State)
   END_RUNG
   // the same network as SCL:
   "DI_Частотник_2_Готов"(input_value := "Частотник (работа) 2",   // "FB_DI"
                          stParamDI := "DI".DI_8,
                          Value => "Conveyor".Conveyor_2.bInRun_Ok_State);
END_REGION

REGION Network 10: Работа чатотника - 3
   RUNG wire#powerrail
      "DI_Частотник_3_Готов"(input_value := "Частотник (работа) 3", stParamDI := "DI".DI_9, Value => "Conveyor".Conveyor_3.bInRun_Ok_State)
   END_RUNG
   // the same network as SCL:
   "DI_Частотник_3_Готов"(input_value := "Частотник (работа) 3",   // "FB_DI"
                          stParamDI := "DI".DI_9,
                          Value => "Conveyor".Conveyor_3.bInRun_Ok_State);
END_REGION

REGION Network 11: Пускатель №1 - включен
   RUNG wire#powerrail
      "DI_Пускатель - 1(вкл)"(input_value := "Пускатель включен 1", stParamDI := "DI".DI_10, Value => "Pumps".Pump_1.bIn_PuskatelState)
   END_RUNG
   // the same network as SCL:
   "DI_Пускатель - 1(вкл)"(input_value := "Пускатель включен 1",   // "FB_DI"
                           stParamDI := "DI".DI_10,
                           Value => "Pumps".Pump_1.bIn_PuskatelState);
END_REGION

REGION Network 12: Пускатель №2 - включен
   RUNG wire#powerrail
      "DI_Пускатель - 2(вкл)"(input_value := "Пускатель включен 2", stParamDI := "DI".DI_11, Value => "Pumps".Pump_2.bIn_PuskatelState)
   END_RUNG
   // the same network as SCL:
   "DI_Пускатель - 2(вкл)"(input_value := "Пускатель включен 2",   // "FB_DI"
                           stParamDI := "DI".DI_11,
                           Value => "Pumps".Pump_2.bIn_PuskatelState);
END_REGION

REGION Network 13: Пускатель №3 - включен
   // Насос - 3
   RUNG wire#powerrail
      "DI_Пускатель - 3(вкл)"(input_value := "Пускатель включен 3", stParamDI := "DI".DI_12, Value => "Pumps".Pump_3.bIn_PuskatelState)
   END_RUNG
   // the same network as SCL:
   "DI_Пускатель - 3(вкл)"(input_value := "Пускатель включен 3",   // "FB_DI"
                           stParamDI := "DI".DI_12,
                           Value => "Pumps".Pump_3.bIn_PuskatelState);
END_REGION

REGION Network 14: Пускатель №4 - включен
   // Насос - 4
   RUNG wire#powerrail
      "DI_Пускатель - 4(вкл)"(input_value := "Пускатель включен 4", stParamDI := "DI".DI_13, Value => "Pumps".Pump_4.bIn_PuskatelState)
   END_RUNG
   // the same network as SCL:
   "DI_Пускатель - 4(вкл)"(input_value := "Пускатель включен 4",   // "FB_DI"
                           stParamDI := "DI".DI_13,
                           Value => "Pumps".Pump_4.bIn_PuskatelState);
END_REGION

REGION Network 15: Пускатель №5 - включен
   // Насос - 5
   RUNG wire#powerrail
      "DI_Пускатель - 5(вкл)"(input_value := "Пускатель включен 5", stParamDI := "DI".DI_14, Value => "Pumps".Pump_5.bIn_PuskatelState)
   END_RUNG
   // the same network as SCL:
   "DI_Пускатель - 5(вкл)"(input_value := "Пускатель включен 5",   // "FB_DI"
                           stParamDI := "DI".DI_14,
                           Value => "Pumps".Pump_5.bIn_PuskatelState);
END_REGION

REGION Network 16: Пускатель №6 - включен
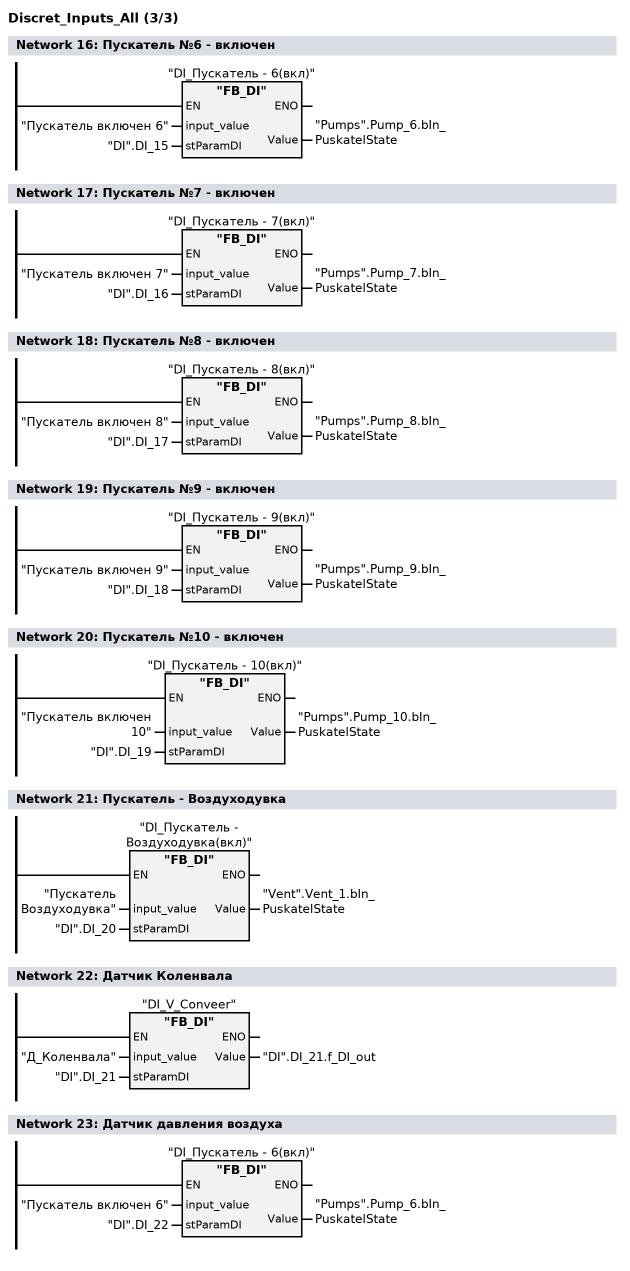
   RUNG wire#powerrail
      "DI_Пускатель - 6(вкл)"(input_value := "Пускатель включен 6", stParamDI := "DI".DI_15, Value => "Pumps".Pump_6.bIn_PuskatelState)
   END_RUNG
   // the same network as SCL:
   "DI_Пускатель - 6(вкл)"(input_value := "Пускатель включен 6",   // "FB_DI"
                           stParamDI := "DI".DI_15,
                           Value => "Pumps".Pump_6.bIn_PuskatelState);
END_REGION

REGION Network 17: Пускатель №7 - включен
   RUNG wire#powerrail
      "DI_Пускатель - 7(вкл)"(input_value := "Пускатель включен 7", stParamDI := "DI".DI_16, Value => "Pumps".Pump_7.bIn_PuskatelState)
   END_RUNG
   // the same network as SCL:
   "DI_Пускатель - 7(вкл)"(input_value := "Пускатель включен 7",   // "FB_DI"
                           stParamDI := "DI".DI_16,
                           Value => "Pumps".Pump_7.bIn_PuskatelState);
END_REGION

REGION Network 18: Пускатель №8 - включен
   RUNG wire#powerrail
      "DI_Пускатель - 8(вкл)"(input_value := "Пускатель включен 8", stParamDI := "DI".DI_17, Value => "Pumps".Pump_8.bIn_PuskatelState)
   END_RUNG
   // the same network as SCL:
   "DI_Пускатель - 8(вкл)"(input_value := "Пускатель включен 8",   // "FB_DI"
                           stParamDI := "DI".DI_17,
                           Value => "Pumps".Pump_8.bIn_PuskatelState);
END_REGION

REGION Network 19: Пускатель №9 - включен
   RUNG wire#powerrail
      "DI_Пускатель - 9(вкл)"(input_value := "Пускатель включен 9", stParamDI := "DI".DI_18, Value => "Pumps".Pump_9.bIn_PuskatelState)
   END_RUNG
   // the same network as SCL:
   "DI_Пускатель - 9(вкл)"(input_value := "Пускатель включен 9",   // "FB_DI"
                           stParamDI := "DI".DI_18,
                           Value => "Pumps".Pump_9.bIn_PuskatelState);
END_REGION

REGION Network 20: Пускатель №10 - включен
   RUNG wire#powerrail
      "DI_Пускатель - 10(вкл)"(input_value := "Пускатель включен 10", stParamDI := "DI".DI_19, Value => "Pumps".Pump_10.bIn_PuskatelState)
   END_RUNG
   // the same network as SCL:
   "DI_Пускатель - 10(вкл)"(input_value := "Пускатель включен 10",   // "FB_DI"
                           stParamDI := "DI".DI_19,
                           Value => "Pumps".Pump_10.bIn_PuskatelState);
END_REGION

REGION Network 21: Пускатель - Воздуходувка
   RUNG wire#powerrail
      "DI_Пускатель - Воздуходувка(вкл)"(input_value := "Пускатель Воздуходувка", stParamDI := "DI".DI_20, Value => "Vent".Vent_1.bIn_PuskatelState)
   END_RUNG
   // the same network as SCL:
   "DI_Пускатель - Воздуходувка(вкл)"(input_value := "Пускатель Воздуходувка",   // "FB_DI"
                           stParamDI := "DI".DI_20,
                           Value => "Vent".Vent_1.bIn_PuskatelState);
END_REGION

REGION Network 22: Датчик Коленвала
   RUNG wire#powerrail
      "DI_V_Conveer"(input_value := "Д_Коленвала", stParamDI := "DI".DI_21, Value => "DI".DI_21.f_DI_out)
   END_RUNG
   // the same network as SCL:
   "DI_V_Conveer"(input_value := "Д_Коленвала", stParamDI := "DI".DI_21, Value => "DI".DI_21.f_DI_out);   // "FB_DI"
END_REGION

REGION Network 23: Датчик давления воздуха
   RUNG wire#powerrail
      "DI_Пускатель - 6(вкл)"(input_value := "Пускатель включен 6", stParamDI := "DI".DI_22, Value => "Pumps".Pump_6.bIn_PuskatelState)
   END_RUNG
   // the same network as SCL:
   "DI_Пускатель - 6(вкл)"(input_value := "Пускатель включен 6",   // "FB_DI"
                           stParamDI := "DI".DI_22,
                           Value => "Pumps".Pump_6.bIn_PuskatelState);
END_REGION
END_FUNCTION

FUNCTION "Конвейера" : Void   // FC9, LAD
{ S7_Optimized_Access := 'TRUE' }
VERSION : 0.1
// Блоки для управления "Конвейерами"
BEGIN

REGION Network 1: Конвейер - 1
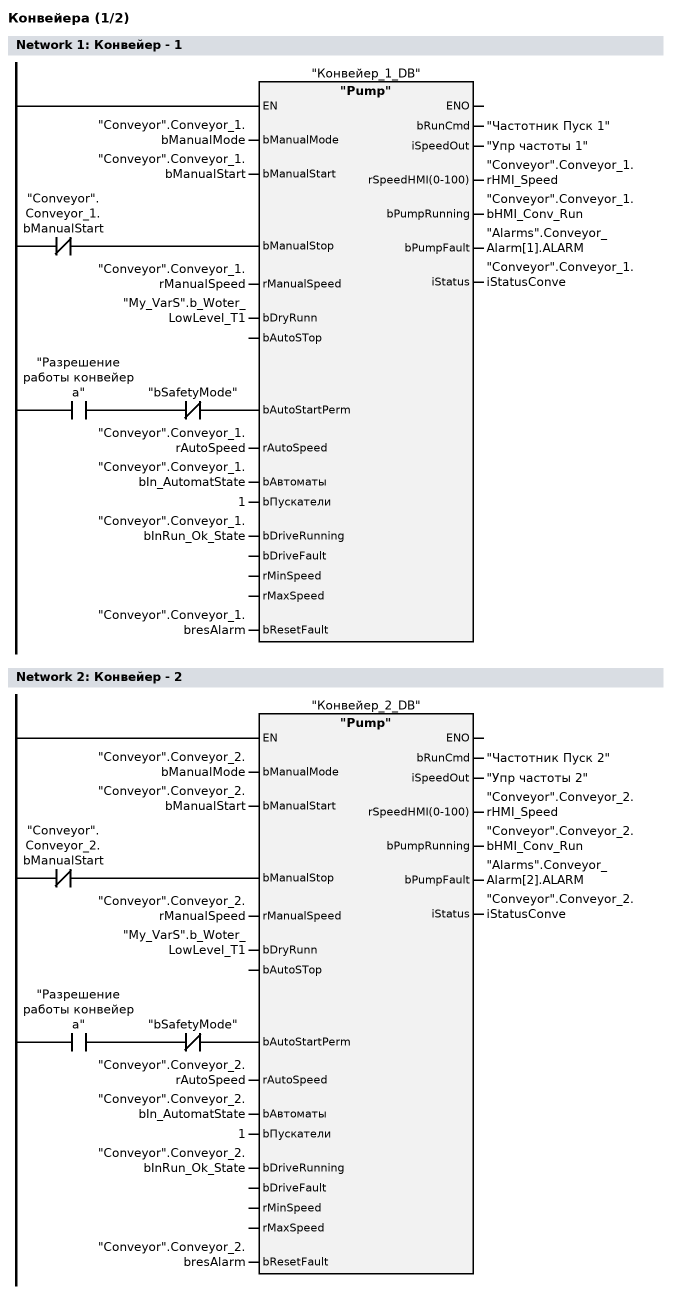
   RUNG wire#powerrail
      "Конвейер_1_DB"(bManualStop := wire#w1, bAutoStartPerm := wire#w2, bManualMode := "Conveyor".Conveyor_1.bManualMode, bManualStart := "Conveyor".Conveyor_1.bManualStart, rManualSpeed := "Conveyor".Conveyor_1.rManualSpeed, bDryRunn := "My_VarS".b_Woter_LowLevel_T1, bAutoSTop :=, rAutoSpeed := "Conveyor".Conveyor_1.rAutoSpeed, bАвтоматы := "Conveyor".Conveyor_1.bIn_AutomatState, bПускатели := 1, bDriveRunning := "Conveyor".Conveyor_1.bInRun_Ok_State, bDriveFault :=, rMinSpeed :=, rMaxSpeed :=, bResetFault := "Conveyor".Conveyor_1.bresAlarm, bRunCmd => "Частотник Пуск 1", iSpeedOut => "Упр частоты 1", "rSpeedHMI(0-100)" => "Conveyor".Conveyor_1.rHMI_Speed, bPumpRunning => "Conveyor".Conveyor_1.bHMI_Conv_Run, bPumpFault => "Alarms".Conveyor_Alarm[1].ALARM, iStatus => "Conveyor".Conveyor_1.iStatusConve)
   END_RUNG
   RUNG wire#powerrail
      I_Contact( "Conveyor".Conveyor_1.bManualStart )
   END_RUNG wire#w1
   RUNG wire#powerrail
      Contact( "Разрешение работы конвейера" )
      I_Contact( "bSafetyMode" )
   END_RUNG wire#w2
   // the same network as SCL:
   "Конвейер_1_DB"(bManualMode := "Conveyor".Conveyor_1.bManualMode,   // "Pump"
                   bManualStart := "Conveyor".Conveyor_1.bManualStart,
                   bManualStop := NOT "Conveyor".Conveyor_1.bManualStart,
                   rManualSpeed := "Conveyor".Conveyor_1.rManualSpeed,
                   bDryRunn := "My_VarS".b_Woter_LowLevel_T1,
                   bAutoStartPerm := "Разрешение работы конвейера" AND NOT "bSafetyMode",
                   rAutoSpeed := "Conveyor".Conveyor_1.rAutoSpeed,
                   bАвтоматы := "Conveyor".Conveyor_1.bIn_AutomatState,
                   bПускатели := 1,
                   bDriveRunning := "Conveyor".Conveyor_1.bInRun_Ok_State,
                   bResetFault := "Conveyor".Conveyor_1.bresAlarm,
                   bRunCmd => "Частотник Пуск 1",
                   iSpeedOut => "Упр частоты 1",
                   "rSpeedHMI(0-100)" => "Conveyor".Conveyor_1.rHMI_Speed,
                   bPumpRunning => "Conveyor".Conveyor_1.bHMI_Conv_Run,
                   bPumpFault => "Alarms".Conveyor_Alarm[1].ALARM,
                   iStatus => "Conveyor".Conveyor_1.iStatusConve);
END_REGION

REGION Network 2: Конвейер - 2
   RUNG wire#powerrail
      "Конвейер_2_DB"(bManualStop := wire#w1, bAutoStartPerm := wire#w2, bManualMode := "Conveyor".Conveyor_2.bManualMode, bManualStart := "Conveyor".Conveyor_2.bManualStart, rManualSpeed := "Conveyor".Conveyor_2.rManualSpeed, bDryRunn := "My_VarS".b_Woter_LowLevel_T1, bAutoSTop :=, rAutoSpeed := "Conveyor".Conveyor_2.rAutoSpeed, bАвтоматы := "Conveyor".Conveyor_2.bIn_AutomatState, bПускатели := 1, bDriveRunning := "Conveyor".Conveyor_2.bInRun_Ok_State, bDriveFault :=, rMinSpeed :=, rMaxSpeed :=, bResetFault := "Conveyor".Conveyor_2.bresAlarm, bRunCmd => "Частотник Пуск 2", iSpeedOut => "Упр частоты 2", "rSpeedHMI(0-100)" => "Conveyor".Conveyor_2.rHMI_Speed, bPumpRunning => "Conveyor".Conveyor_2.bHMI_Conv_Run, bPumpFault => "Alarms".Conveyor_Alarm[2].ALARM, iStatus => "Conveyor".Conveyor_2.iStatusConve)
   END_RUNG
   RUNG wire#powerrail
      I_Contact( "Conveyor".Conveyor_2.bManualStart )
   END_RUNG wire#w1
   RUNG wire#powerrail
      Contact( "Разрешение работы конвейера" )
      I_Contact( "bSafetyMode" )
   END_RUNG wire#w2
   // the same network as SCL:
   "Конвейер_2_DB"(bManualMode := "Conveyor".Conveyor_2.bManualMode,   // "Pump"
                   bManualStart := "Conveyor".Conveyor_2.bManualStart,
                   bManualStop := NOT "Conveyor".Conveyor_2.bManualStart,
                   rManualSpeed := "Conveyor".Conveyor_2.rManualSpeed,
                   bDryRunn := "My_VarS".b_Woter_LowLevel_T1,
                   bAutoStartPerm := "Разрешение работы конвейера" AND NOT "bSafetyMode",
                   rAutoSpeed := "Conveyor".Conveyor_2.rAutoSpeed,
                   bАвтоматы := "Conveyor".Conveyor_2.bIn_AutomatState,
                   bПускатели := 1,
                   bDriveRunning := "Conveyor".Conveyor_2.bInRun_Ok_State,
                   bResetFault := "Conveyor".Conveyor_2.bresAlarm,
                   bRunCmd => "Частотник Пуск 2",
                   iSpeedOut => "Упр частоты 2",
                   "rSpeedHMI(0-100)" => "Conveyor".Conveyor_2.rHMI_Speed,
                   bPumpRunning => "Conveyor".Conveyor_2.bHMI_Conv_Run,
                   bPumpFault => "Alarms".Conveyor_Alarm[2].ALARM,
                   iStatus => "Conveyor".Conveyor_2.iStatusConve);
END_REGION

REGION Network 3: Конвейер - 3
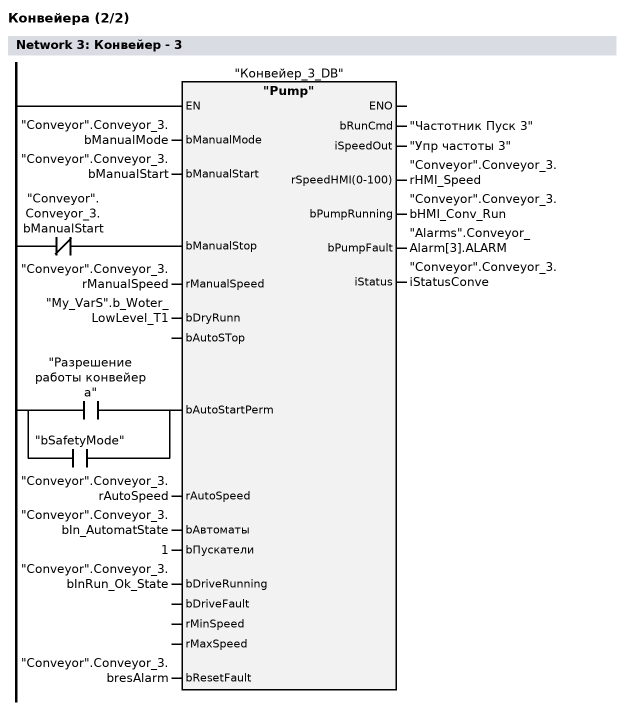
   RUNG wire#powerrail
      "Конвейер_3_DB"(bManualStop := wire#w1, bAutoStartPerm := wire#w2, bManualMode := "Conveyor".Conveyor_3.bManualMode, bManualStart := "Conveyor".Conveyor_3.bManualStart, rManualSpeed := "Conveyor".Conveyor_3.rManualSpeed, bDryRunn := "My_VarS".b_Woter_LowLevel_T1, bAutoSTop :=, rAutoSpeed := "Conveyor".Conveyor_3.rAutoSpeed, bАвтоматы := "Conveyor".Conveyor_3.bIn_AutomatState, bПускатели := 1, bDriveRunning := "Conveyor".Conveyor_3.bInRun_Ok_State, bDriveFault :=, rMinSpeed :=, rMaxSpeed :=, bResetFault := "Conveyor".Conveyor_3.bresAlarm, bRunCmd => "Частотник Пуск 3", iSpeedOut => "Упр частоты 3", "rSpeedHMI(0-100)" => "Conveyor".Conveyor_3.rHMI_Speed, bPumpRunning => "Conveyor".Conveyor_3.bHMI_Conv_Run, bPumpFault => "Alarms".Conveyor_Alarm[3].ALARM, iStatus => "Conveyor".Conveyor_3.iStatusConve)
   END_RUNG
   RUNG wire#powerrail
      I_Contact( "Conveyor".Conveyor_3.bManualStart )
   END_RUNG wire#w1
   RUNG wire#powerrail
      Contact( "Разрешение работы конвейера" )
   END_RUNG wire#w2
   RUNG wire#powerrail
      Contact( "bSafetyMode" )
   END_RUNG wire#w2
   // the same network as SCL:
   "Конвейер_3_DB"(bManualMode := "Conveyor".Conveyor_3.bManualMode,   // "Pump"
                   bManualStart := "Conveyor".Conveyor_3.bManualStart,
                   bManualStop := NOT "Conveyor".Conveyor_3.bManualStart,
                   rManualSpeed := "Conveyor".Conveyor_3.rManualSpeed,
                   bDryRunn := "My_VarS".b_Woter_LowLevel_T1,
                   bAutoStartPerm := "Разрешение работы конвейера" OR "bSafetyMode",
                   rAutoSpeed := "Conveyor".Conveyor_3.rAutoSpeed,
                   bАвтоматы := "Conveyor".Conveyor_3.bIn_AutomatState,
                   bПускатели := 1,
                   bDriveRunning := "Conveyor".Conveyor_3.bInRun_Ok_State,
                   bResetFault := "Conveyor".Conveyor_3.bresAlarm,
                   bRunCmd => "Частотник Пуск 3",
                   iSpeedOut => "Упр частоты 3",
                   "rSpeedHMI(0-100)" => "Conveyor".Conveyor_3.rHMI_Speed,
                   bPumpRunning => "Conveyor".Conveyor_3.bHMI_Conv_Run,
                   bPumpFault => "Alarms".Conveyor_Alarm[3].ALARM,
                   iStatus => "Conveyor".Conveyor_3.iStatusConve);
END_REGION
END_FUNCTION

FUNCTION "Вентилятор" : Void   // FC10, LAD
{ S7_Optimized_Access := 'TRUE' }
VERSION : 0.1
// Управление вентилятором
BEGIN

REGION Network 1: Вентилятор
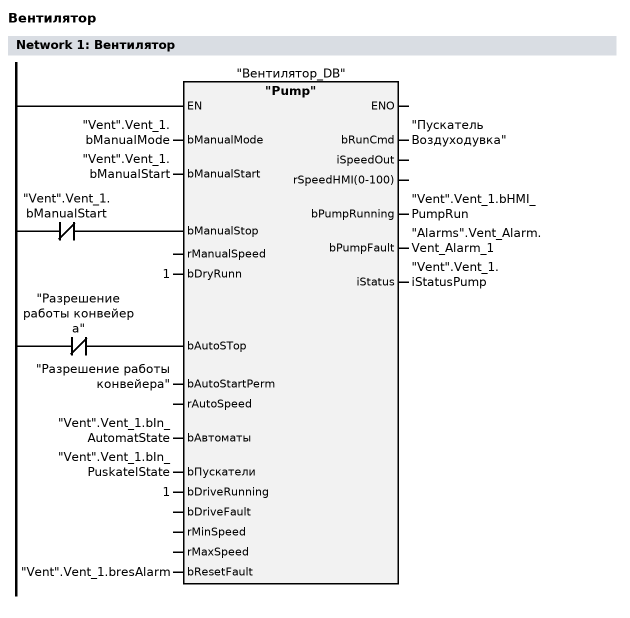
   RUNG wire#powerrail
      "Вентилятор_DB"(bManualStop := wire#w1, bAutoSTop := wire#w2, bManualMode := "Vent".Vent_1.bManualMode, bManualStart := "Vent".Vent_1.bManualStart, rManualSpeed :=, bDryRunn := 1, bAutoStartPerm := "Разрешение работы конвейера", rAutoSpeed :=, bАвтоматы := "Vent".Vent_1.bIn_AutomatState, bПускатели := "Vent".Vent_1.bIn_PuskatelState, bDriveRunning := 1, bDriveFault :=, rMinSpeed :=, rMaxSpeed :=, bResetFault := "Vent".Vent_1.bresAlarm, bRunCmd => "Пускатель Воздуходувка", iSpeedOut =>, "rSpeedHMI(0-100)" =>, bPumpRunning => "Vent".Vent_1.bHMI_PumpRun, bPumpFault => "Alarms".Vent_Alarm.Vent_Alarm_1, iStatus => "Vent".Vent_1.iStatusPump)
   END_RUNG
   RUNG wire#powerrail
      I_Contact( "Vent".Vent_1.bManualStart )
   END_RUNG wire#w1
   RUNG wire#powerrail
      I_Contact( "Разрешение работы конвейера" )
   END_RUNG wire#w2
   // the same network as SCL:
   "Вентилятор_DB"(bManualMode := "Vent".Vent_1.bManualMode,   // "Pump"
                   bManualStart := "Vent".Vent_1.bManualStart,
                   bManualStop := NOT "Vent".Vent_1.bManualStart,
                   bDryRunn := 1,
                   bAutoSTop := NOT "Разрешение работы конвейера",
                   bAutoStartPerm := "Разрешение работы конвейера",
                   bАвтоматы := "Vent".Vent_1.bIn_AutomatState,
                   bПускатели := "Vent".Vent_1.bIn_PuskatelState,
                   bDriveRunning := 1,
                   bResetFault := "Vent".Vent_1.bresAlarm,
                   bRunCmd => "Пускатель Воздуходувка",
                   bPumpRunning => "Vent".Vent_1.bHMI_PumpRun,
                   bPumpFault => "Alarms".Vent_Alarm.Vent_Alarm_1,
                   iStatus => "Vent".Vent_1.iStatusPump);
END_REGION
END_FUNCTION

FUNCTION "Работа клапана подпидки" : Void   // FC11, LAD
{ S7_Optimized_Access := 'TRUE' }
VERSION : 0.1
BEGIN

REGION Network 1: Бак 1
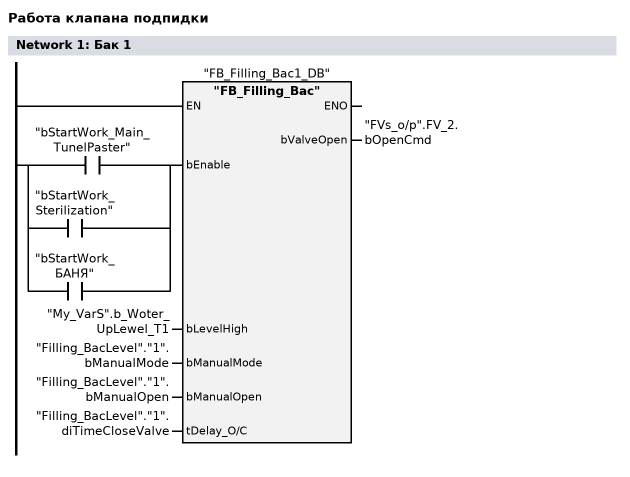
   RUNG wire#powerrail
      "FB_Filling_Bac1_DB"(bEnable := wire#w1, bLevelHigh := "My_VarS".b_Woter_UpLewel_T1, bManualMode := "Filling_BacLevel"."1".bManualMode, bManualOpen := "Filling_BacLevel"."1".bManualOpen, "tDelay_O/C" := "Filling_BacLevel"."1".diTimeCloseValve, bValveOpen => "FVs_o/p".FV_2.bOpenCmd)
   END_RUNG
   RUNG wire#powerrail
      Contact( "bStartWork_Main_TunelPaster" )
   END_RUNG wire#w1
   RUNG wire#powerrail
      Contact( "bStartWork_Sterilization" )
   END_RUNG wire#w1
   RUNG wire#powerrail
      Contact( "bStartWork_БАНЯ" )
   END_RUNG wire#w1
   // the same network as SCL:
   "FB_Filling_Bac1_DB"(bEnable := "bStartWork_Main_TunelPaster" OR "bStartWork_Sterilization" OR "bStartWork_БАНЯ",   // "FB_Filling_Bac"
                        bLevelHigh := "My_VarS".b_Woter_UpLewel_T1,
                        bManualMode := "Filling_BacLevel"."1".bManualMode,
                        bManualOpen := "Filling_BacLevel"."1".bManualOpen,
                        "tDelay_O/C" := "Filling_BacLevel"."1".diTimeCloseValve,
                        bValveOpen => "FVs_o/p".FV_2.bOpenCmd);
END_REGION
END_FUNCTION

FUNCTION "Все в Авто" : Void   // FC12, SCL
{ S7_Optimized_Access := 'TRUE' }
VERSION : 0.1
   VAR_TEMP
      fTrig_All_Auto : Bool;   // Фронт нажития кнопки все в авто
   END_VAR
BEGIN

   //Отлавливаем фронт нажатия клавиши все в авто
   "R_trig_All_Auto"(In:="bAllAuto",
                     Q=>#fTrig_All_Auto);

   //Сбрасываем все ручное в автоматический режим
   //
   IF #fTrig_All_Auto THEN

       //симуляция датчиков аналоговых
       "AI_DB".AI_1.bSimulate := FALSE;
       "AI_DB".AI_2.bSimulate := FALSE;
       "AI_DB".AI_3.bSimulate := FALSE;
       "AI_DB".AI_4.bSimulate := FALSE;
       "AI_DB".AI_5.bSimulate := FALSE;
       "AI_DB".AI_6.bSimulate := FALSE;
       "AI_DB".AI_7.bSimulate := FALSE;

       "AI_DB"."AI_4-20_1".bSimulate := FALSE;
       "AI_DB"."AI_4-20_2".bSimulate := FALSE;
       "AI_DB"."AI_4-20_3".bSimulate := FALSE;

       //Управление конвейером в ручном режиме
       "Conveyor".Conveyor_1.bManualMode := FALSE;
       "Conveyor".Conveyor_2.bManualMode := FALSE;
       "Conveyor".Conveyor_3.bManualMode := FALSE;
       "Conveyor".Conveyor_4.bManualMode := FALSE;

       //Управление баками наполнения
       "Filling_BacLevel"."1".bManualMode := FALSE;


       //Управление FV - Open/Close
       "FVs_o/p".FV_4.bManualMode := FALSE;
       "FVs_o/p".FV_5.bManualMode := FALSE;
       "FVs_o/p".FV_1.bManualMode := FALSE;


       //Управление FV - Regul 
       "FVs_Regul".FV_Regul_1.bHMI_ManualMode := FALSE;
       "FVs_Regul".FV_Regul_2.bHMI_ManualMode := FALSE;
       "FVs_Regul".FV_Regul_3.bHMI_ManualMode := FALSE;
       "FVs_Regul".FV_Regul_4.bHMI_ManualMode := FALSE;
       "FVs_Regul".FV_Regul_7.bHMI_ManualMode := FALSE;



       //Управление Pumps
       "Pumps".Pump_1.bManualMode := FALSE;
       "Pumps".Pump_2.bManualMode := FALSE;
       "Pumps".Pump_3.bManualMode := FALSE;
       "Pumps".Pump_4.bManualMode := FALSE;
       "Pumps".Pump_5.bManualMode := FALSE;
       "Pumps".Pump_6.bManualMode := FALSE;
       "Pumps".Pump_7.bManualMode := FALSE;


       //Управление Vent
       "Vent".Vent_1.bManualMode := FALSE;

       //DI
       (*
       "DI".DI_0.bSimulation := FALSE;
       "DI".DI_1.bSimulation := FALSE;
       "DI".DI_2.bSimulation := FALSE;
       "DI".DI_3.bSimulation := FALSE;
       "DI".DI_4.bSimulation := FALSE;
       "DI".DI_5.bSimulation := FALSE;
       "DI".DI_6.bSimulation := FALSE;
       "DI".DI_7.bSimulation := FALSE;
       "DI".DI_8.bSimulation := FALSE;
       "DI".DI_9.bSimulation := FALSE;
       "DI".DI_10.bSimulation := FALSE;
       "DI".DI_11.bSimulation := FALSE;
       "DI".DI_12.bSimulation := FALSE;
       "DI".DI_13.bSimulation := FALSE;
       "DI".DI_14.bSimulation := FALSE;
       "DI".DI_15.bSimulation := FALSE;
       "DI".DI_16.bSimulation := FALSE;
       "DI".DI_17.bSimulation := FALSE;
       "DI".DI_18.bSimulation := FALSE;
       "DI".DI_19.bSimulation := FALSE;
       "DI".DI_20.bSimulation := FALSE;
       "DI".DI_21.bSimulation := FALSE;
       "DI".DI_22.bSimulation := FALSE;
       "DI".DI_23.bSimulation := FALSE;
       "DI".DI_24.bSimulation := FALSE;
       "DI".DI_25.bSimulation := FALSE;
       "DI".DI_26.bSimulation := FALSE;
       "DI".DI_27.bSimulation := FALSE;
       "DI".DI_28.bSimulation := FALSE;
       "DI".DI_29.bSimulation := FALSE;
      *)
   END_IF;
END_FUNCTION

FUNCTION "RestetAlarms" : Void   // FC13, SCL
{ S7_Optimized_Access := 'TRUE' }
VERSION : 0.1
BEGIN
   IF "bResetCommon" THEN
       //Сброс аварий насосов
       "Pumps".Pump_1.bresAlarm := TRUE;
       "Pumps".Pump_2.bresAlarm := TRUE;
       "Pumps".Pump_3.bresAlarm := TRUE;
       "Pumps".Pump_4.bresAlarm := TRUE;
       "Pumps".Pump_5.bresAlarm := TRUE;
       "Pumps".Pump_6.bresAlarm := TRUE;
       "Pumps".Pump_7.bresAlarm := TRUE;

       //Сброс аварий конвейера
       "Conveyor".Conveyor_1.bresAlarm := TRUE;
       "Conveyor".Conveyor_2.bresAlarm := TRUE;
       "Conveyor".Conveyor_3.bresAlarm := TRUE;
       "Conveyor".Conveyor_4.bresAlarm := TRUE;

       //Сброс аварий вентилятор
       "Vent".Vent_1.bresAlarm := TRUE;

       //Сброс аварий клапана
       "FVs_o/p".FV_4.bResetAlarm := TRUE;
       "FVs_o/p".FV_5.bResetAlarm := TRUE;
       "FVs_o/p".FV_1.bResetAlarm := TRUE;



   ELSE
       //Сброс аварий насосов
       "Pumps".Pump_1.bresAlarm := False;
       "Pumps".Pump_2.bresAlarm := False;
       "Pumps".Pump_3.bresAlarm := False;
       "Pumps".Pump_4.bresAlarm := False;
       "Pumps".Pump_5.bresAlarm := False;
       "Pumps".Pump_6.bresAlarm := False;
       "Pumps".Pump_7.bresAlarm := False;

       //Сброс аварий конвейера
       "Conveyor".Conveyor_1.bresAlarm := False;
       "Conveyor".Conveyor_2.bresAlarm := False;
       "Conveyor".Conveyor_3.bresAlarm := False;
       "Conveyor".Conveyor_4.bresAlarm := False;

       //Сброс аварий вентилятор
       "Vent".Vent_1.bresAlarm := FALSE;

       //Сброс аварий клапана
       "FVs_o/p".FV_4.bResetAlarm := False;
       "FVs_o/p".FV_5.bResetAlarm := False;
       "FVs_o/p".FV_1.bResetAlarm := False;


   END_IF;
END_FUNCTION

FUNCTION "Зоны Стерилизации_Контроль" : Void   // FC14, LAD
{ S7_Optimized_Access := 'TRUE' }
VERSION : 0.1
BEGIN

REGION Network 1: Зона 1
   // Зона 1
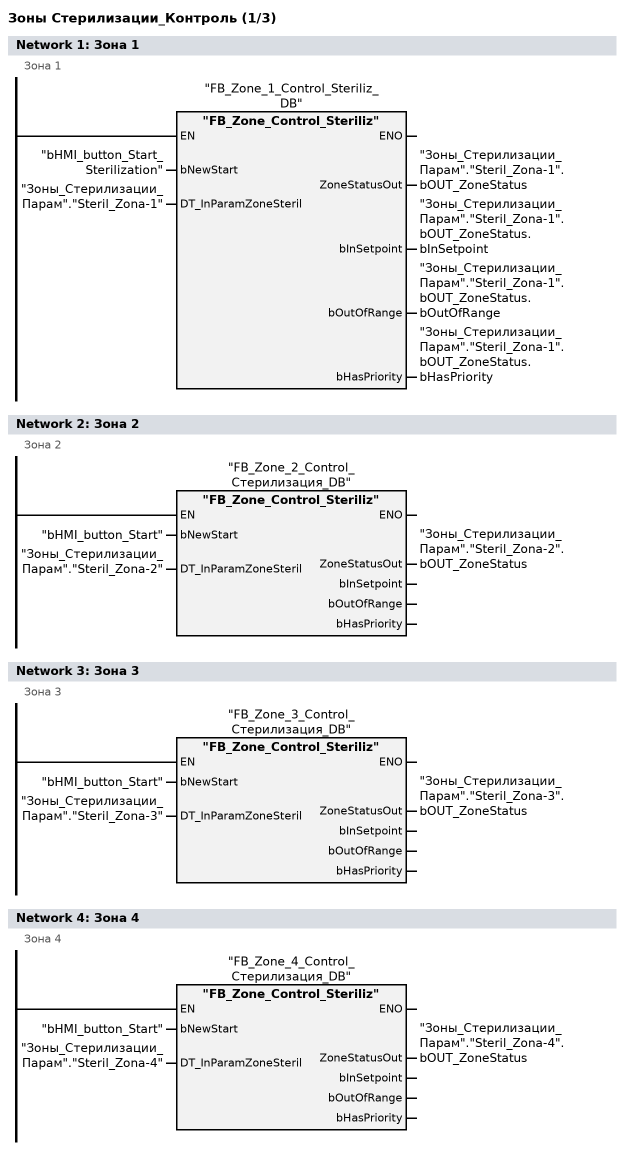
   RUNG wire#powerrail
      "FB_Zone_1_Control_Steriliz_DB"(bNewStart := "bHMI_button_Start_Sterilization", DT_InParamZoneSteril := "Зоны_Стерилизации_Парам"."Steril_Zona-1", ZoneStatusOut => "Зоны_Стерилизации_Парам"."Steril_Zona-1".bOUT_ZoneStatus, bInSetpoint => "Зоны_Стерилизации_Парам"."Steril_Zona-1".bOUT_ZoneStatus.bInSetpoint, bOutOfRange => "Зоны_Стерилизации_Парам"."Steril_Zona-1".bOUT_ZoneStatus.bOutOfRange, bHasPriority => "Зоны_Стерилизации_Парам"."Steril_Zona-1".bOUT_ZoneStatus.bHasPriority)
   END_RUNG
   // the same network as SCL:
   "FB_Zone_1_Control_Steriliz_DB"(bNewStart := "bHMI_button_Start_Sterilization",   // "FB_Zone_Control_Steriliz"
                           DT_InParamZoneSteril := "Зоны_Стерилизации_Парам"."Steril_Zona-1",
                           ZoneStatusOut => "Зоны_Стерилизации_Парам"."Steril_Zona-1".bOUT_ZoneStatus,
                           bInSetpoint => "Зоны_Стерилизации_Парам"."Steril_Zona-1".bOUT_ZoneStatus.bInSetpoint,
                           bOutOfRange => "Зоны_Стерилизации_Парам"."Steril_Zona-1".bOUT_ZoneStatus.bOutOfRange,
                           bHasPriority => "Зоны_Стерилизации_Парам"."Steril_Zona-1".bOUT_ZoneStatus.bHasPriority);
END_REGION

REGION Network 2: Зона 2
   // Зона 2
   RUNG wire#powerrail
      "FB_Zone_2_Control_Стерилизация_DB"(bNewStart := "bHMI_button_Start", DT_InParamZoneSteril := "Зоны_Стерилизации_Парам"."Steril_Zona-2", ZoneStatusOut => "Зоны_Стерилизации_Парам"."Steril_Zona-2".bOUT_ZoneStatus, bInSetpoint =>, bOutOfRange =>, bHasPriority =>)
   END_RUNG
   // the same network as SCL:
   "FB_Zone_2_Control_Стерилизация_DB"(bNewStart := "bHMI_button_Start",   // "FB_Zone_Control_Steriliz"
                           DT_InParamZoneSteril := "Зоны_Стерилизации_Парам"."Steril_Zona-2",
                           ZoneStatusOut => "Зоны_Стерилизации_Парам"."Steril_Zona-2".bOUT_ZoneStatus);
END_REGION

REGION Network 3: Зона 3
   // Зона 3
   RUNG wire#powerrail
      "FB_Zone_3_Control_Стерилизация_DB"(bNewStart := "bHMI_button_Start", DT_InParamZoneSteril := "Зоны_Стерилизации_Парам"."Steril_Zona-3", ZoneStatusOut => "Зоны_Стерилизации_Парам"."Steril_Zona-3".bOUT_ZoneStatus, bInSetpoint =>, bOutOfRange =>, bHasPriority =>)
   END_RUNG
   // the same network as SCL:
   "FB_Zone_3_Control_Стерилизация_DB"(bNewStart := "bHMI_button_Start",   // "FB_Zone_Control_Steriliz"
                           DT_InParamZoneSteril := "Зоны_Стерилизации_Парам"."Steril_Zona-3",
                           ZoneStatusOut => "Зоны_Стерилизации_Парам"."Steril_Zona-3".bOUT_ZoneStatus);
END_REGION

REGION Network 4: Зона 4
   // Зона 4
   RUNG wire#powerrail
      "FB_Zone_4_Control_Стерилизация_DB"(bNewStart := "bHMI_button_Start", DT_InParamZoneSteril := "Зоны_Стерилизации_Парам"."Steril_Zona-4", ZoneStatusOut => "Зоны_Стерилизации_Парам"."Steril_Zona-4".bOUT_ZoneStatus, bInSetpoint =>, bOutOfRange =>, bHasPriority =>)
   END_RUNG
   // the same network as SCL:
   "FB_Zone_4_Control_Стерилизация_DB"(bNewStart := "bHMI_button_Start",   // "FB_Zone_Control_Steriliz"
                           DT_InParamZoneSteril := "Зоны_Стерилизации_Парам"."Steril_Zona-4",
                           ZoneStatusOut => "Зоны_Стерилизации_Парам"."Steril_Zona-4".bOUT_ZoneStatus);
END_REGION

REGION Network 5: Зона 5
   // Зона 5
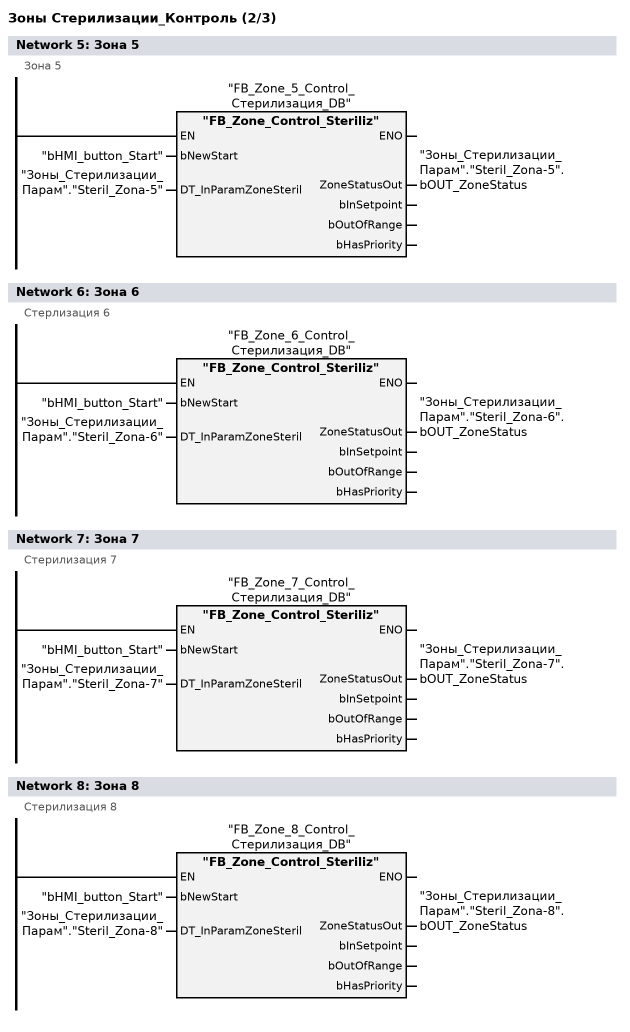
   RUNG wire#powerrail
      "FB_Zone_5_Control_Стерилизация_DB"(bNewStart := "bHMI_button_Start", DT_InParamZoneSteril := "Зоны_Стерилизации_Парам"."Steril_Zona-5", ZoneStatusOut => "Зоны_Стерилизации_Парам"."Steril_Zona-5".bOUT_ZoneStatus, bInSetpoint =>, bOutOfRange =>, bHasPriority =>)
   END_RUNG
   // the same network as SCL:
   "FB_Zone_5_Control_Стерилизация_DB"(bNewStart := "bHMI_button_Start",   // "FB_Zone_Control_Steriliz"
                           DT_InParamZoneSteril := "Зоны_Стерилизации_Парам"."Steril_Zona-5",
                           ZoneStatusOut => "Зоны_Стерилизации_Парам"."Steril_Zona-5".bOUT_ZoneStatus);
END_REGION

REGION Network 6: Зона 6
   // Стерлизация 6
   RUNG wire#powerrail
      "FB_Zone_6_Control_Стерилизация_DB"(bNewStart := "bHMI_button_Start", DT_InParamZoneSteril := "Зоны_Стерилизации_Парам"."Steril_Zona-6", ZoneStatusOut => "Зоны_Стерилизации_Парам"."Steril_Zona-6".bOUT_ZoneStatus, bInSetpoint =>, bOutOfRange =>, bHasPriority =>)
   END_RUNG
   // the same network as SCL:
   "FB_Zone_6_Control_Стерилизация_DB"(bNewStart := "bHMI_button_Start",   // "FB_Zone_Control_Steriliz"
                           DT_InParamZoneSteril := "Зоны_Стерилизации_Парам"."Steril_Zona-6",
                           ZoneStatusOut => "Зоны_Стерилизации_Парам"."Steril_Zona-6".bOUT_ZoneStatus);
END_REGION

REGION Network 7: Зона 7
   // Стерилизация 7
   RUNG wire#powerrail
      "FB_Zone_7_Control_Стерилизация_DB"(bNewStart := "bHMI_button_Start", DT_InParamZoneSteril := "Зоны_Стерилизации_Парам"."Steril_Zona-7", ZoneStatusOut => "Зоны_Стерилизации_Парам"."Steril_Zona-7".bOUT_ZoneStatus, bInSetpoint =>, bOutOfRange =>, bHasPriority =>)
   END_RUNG
   // the same network as SCL:
   "FB_Zone_7_Control_Стерилизация_DB"(bNewStart := "bHMI_button_Start",   // "FB_Zone_Control_Steriliz"
                           DT_InParamZoneSteril := "Зоны_Стерилизации_Парам"."Steril_Zona-7",
                           ZoneStatusOut => "Зоны_Стерилизации_Парам"."Steril_Zona-7".bOUT_ZoneStatus);
END_REGION

REGION Network 8: Зона 8
   // Стерилизация 8
   RUNG wire#powerrail
      "FB_Zone_8_Control_Стерилизация_DB"(bNewStart := "bHMI_button_Start", DT_InParamZoneSteril := "Зоны_Стерилизации_Парам"."Steril_Zona-8", ZoneStatusOut => "Зоны_Стерилизации_Парам"."Steril_Zona-8".bOUT_ZoneStatus, bInSetpoint =>, bOutOfRange =>, bHasPriority =>)
   END_RUNG
   // the same network as SCL:
   "FB_Zone_8_Control_Стерилизация_DB"(bNewStart := "bHMI_button_Start",   // "FB_Zone_Control_Steriliz"
                           DT_InParamZoneSteril := "Зоны_Стерилизации_Парам"."Steril_Zona-8",
                           ZoneStatusOut => "Зоны_Стерилизации_Парам"."Steril_Zona-8".bOUT_ZoneStatus);
END_REGION

REGION Network 9: Зона 9
   // Стерилизация 9
